// TIA Portal project "SepDuplo" (V16)

(* hardware
DEVICE "S71500/ET200MP station_1"  S7-1500 station
   slot 0: "Rail_0"  Rack  6ES7 590-1***0-0AA0
   slot 1: "PLC_1"  CPU 1512C-1 PN  6ES7 512-1CK00-0AB0  V2.8
      slot 3: "CPU display_1"  6ES7591-1AA00-0AA0
      slot 32768: "PROFINET interface_1"  X1
         slot 32769: "Port_1"  X1 P1
         slot 32770: "Port_2"  X1 P2
      slot 34817: "Virtual CP interface port_1"  Virtual CP interface port  Virtual CP interface port
*)

// ===== PLC "PLC_1"  CPU 1512C-1 PN =====

VAR_GLOBAL   // PLC tag table "Default tag table"
   "alwaysFalse" AT %M0.0 : Bool;
END_VAR

VAR_GLOBAL   // PLC tag table "E_N_Controlavel"
   "FIO_S3" AT %M5.3 : Bool;
   "FIO_PA1" AT %M5.1 : Bool;
   "FIO_PV1" AT %M5.0 : Bool;
   "FIO_S4" AT %M5.5 : Bool;
   "FIO_AT1_Fwd" AT %M5.6 : Bool;
   "FIO_AT1_Rev" AT %M5.7 : Bool;
   "FIO_PA2" AT %M6.0 : Bool;
   "FIO_PV2" AT %M6.1 : Bool;
   "FIO_S5" AT %M6.2 : Bool;
   "FIO_S6" AT %M6.3 : Bool;
   "FIO_AT2_Fwd" AT %M6.4 : Bool;
   "FIO_AT2_Rev" AT %M6.5 : Bool;
END_VAR

VAR_GLOBAL   // PLC tag table "Saidas"
   "FIO_Atuador1" AT %M10.0 : Bool;
   "FIO_Esteira1" AT %M10.1 : Bool;
   "FIO_Esteira2" AT %M10.2 : Bool;
   "FIO_Esteira3" AT %M10.3 : Bool;
   "FIO_Esteira4" AT %M10.4 : Bool;
   "FIO_Atuador2" AT %M10.5 : Bool;
END_VAR

DATA_BLOCK "Eventos"   // DB1
{ S7_Optimized_Access := 'TRUE' }
VERSION : 0.1
   VAR
      PV1_Ev : Bool;
      PA1_Ev : Bool;
      PV2_Ev : Bool;
      PA2_Ev : Bool;
      S3_On_Ev : Bool;
      S3_On_Mirror : Bool;
      S3_Off_Ev : Bool;
      S4_On_Ev : Bool;
      S4_On_Mirror : Bool;
      S4_Off_Ev : Bool;
      AT1_Off_Ev : Bool;
      AT2_Off_Ev : Bool;
      S5_Off_Ev : Bool;
      S6_Off_Ev : Bool;
      AT1_On_Ev : Bool;
      AT2_On_Ev : Bool;
      E1_On_Ev : Bool;
      E1_Off_Ev : Bool;
      E2_On_Ev : Bool;
      E2_Off_Ev : Bool;
      E3_On_Ev : Bool;
      E3_Off_Ev : Bool;
      E4_On_Ev : Bool;
      E4_Off_Ev : Bool;
   END_VAR
BEGIN
END_DATA_BLOCK

DATA_BLOCK "BitsAuxiliares"   // DB2
{ S7_Optimized_Access := 'TRUE' }
VERSION : 0.1
   VAR
      Aux1 : Bool;
      Aux2 : Bool;
      Aux3 : Bool;
      Aux4 : Bool;
      Aux5 : Bool;
      Aux6 : Bool;
      Aux7 : Bool;
      Aux8 : Bool;
      Aux9 : Bool;
      Aux10 : Bool;
      Aux11 : Bool;
      Aux12 : Bool;
   END_VAR
BEGIN
END_DATA_BLOCK

DATA_BLOCK "EstadosSP"   // DB3
{ S7_Optimized_Access := 'TRUE' }
VERSION : 0.1
   VAR
      GS1_1 : Bool := true;
      GS1_2 : Bool;
      GS1_3 : Bool;
      GS2_1 : Bool := true;
      GS2_2 : Bool;
      GS2_3 : Bool;
      GAT1_1 : Bool := true;
      GAT1_2 : Bool;
      GAT2_1 : Bool := true;
      GAT2_2 : Bool;
      GE1_1 : Bool := true;
      GE1_2 : Bool;
      GE2_1 : Bool := true;
      GE2_2 : Bool;
      GE3_1 : Bool := true;
      GE3_2 : Bool;
      GE4_1 : Bool := true;
      GE4_2 : Bool;
      GS5_1 : Bool := true;
      GS6_1 : Bool := true;
   END_VAR
BEGIN
END_DATA_BLOCK

DATA_BLOCK "EstadosSup"   // DB4
{ S7_Optimized_Access := 'TRUE' }
VERSION : 0.1
   VAR
      Sup1_1 : Bool := true;
      Sup1_2 : Bool;
      Sup2_1 : Bool := true;
      Sup2_2 : Bool;
      Sup3_1 : Bool := true;
      Sup3_2 : Bool;
      Sup3_3 : Bool;
      Sup3_4 : Bool;
      Sup4_1 : Bool := true;
      Sup4_2 : Bool;
      Sup4_3 : Bool;
      Sup4_4 : Bool;
      Sup5_1 : Bool := true;
      Sup5_2 : Bool;
      Sup6_1 : Bool := true;
      Sup6_2 : Bool;
      Sup7_1 : Bool := true;
      Sup7_2 : Bool;
      Sup7_3 : Bool;
      Sup8_1 : Bool := true;
      Sup8_2 : Bool;
      Sup8_3 : Bool;
      Sup9_1 : Bool := true;
      Sup9_2 : Bool;
      Sup10_1 : Bool := true;
      Sup10_2 : Bool;
      Sup11_1 : Bool := true;
      Sup11_2 : Bool;
      Sup12_1 : Bool := true;
      Sup12_2 : Bool;
      Sup13_1 : Bool := true;
      Sup13_2 : Bool;
      Sup13_3 : Bool;
      Sup13_4 : Bool;
      Sup13_5 : Bool;
      Sup13_6 : Bool;
      Sup13_7 : Bool;
      Sup13_8 : Bool;
      Sup13_9 : Bool;
      Sup14_1 : Bool := true;
      Sup14_2 : Bool;
      Sup15_1 : Bool := true;
      Sup15_2 : Bool;
   END_VAR
BEGIN
END_DATA_BLOCK

DATA_BLOCK "Des_Eventos"   // DB5
{ S7_Optimized_Access := 'TRUE' }
VERSION : 0.1
   VAR
      d_AT1_On : Bool;
      d_AT2_On : Bool;
      d_E1_On : Bool;
      d_E1_Off : Bool;
      d_E2_On : Bool;
      d_E2_Off : Bool;
      d_E3_On : Bool;
      d_E3_Off : Bool;
      d_E4_On : Bool;
      d_E4_Off : Bool;
   END_VAR
BEGIN
END_DATA_BLOCK

FUNCTION "LeituraEntradas" : Void   // FC2, LAD
TITLE = Leitura das entradas dos eventos não controláveis
{ S7_Optimized_Access := 'TRUE' }
VERSION : 0.1
   VAR_TEMP   // added for the SCL form of the ladder/FBD networks
      _w1 : Bool;
   END_VAR
BEGIN

REGION Network 1: Leitura peça verde 1
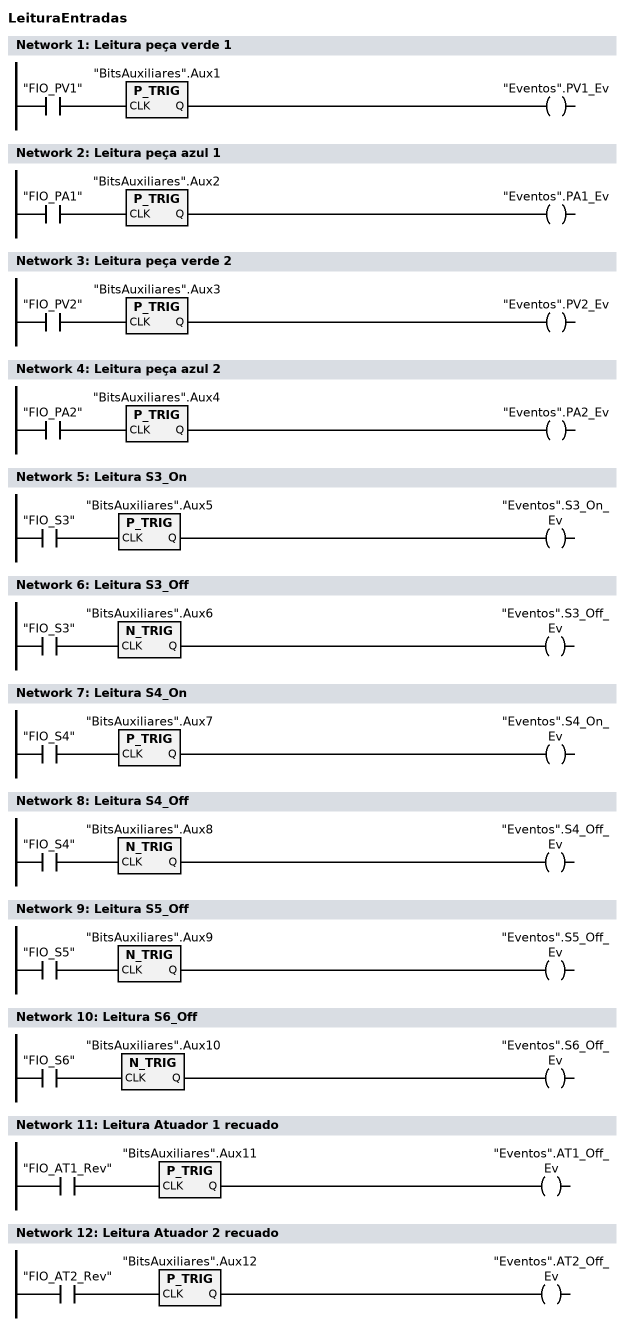
   RUNG wire#powerrail
      Contact( "FIO_PV1" )
      P_Trig( "BitsAuxiliares".Aux1 )
      Coil( "Eventos".PV1_Ev )
   END_RUNG
   // the same network as SCL:
   #_w1 := "FIO_PV1" AND NOT "BitsAuxiliares".Aux1;   // rising edge
   "BitsAuxiliares".Aux1 := "FIO_PV1";
   "Eventos".PV1_Ev := #_w1;
END_REGION

REGION Network 2: Leitura peça azul 1
   RUNG wire#powerrail
      Contact( "FIO_PA1" )
      P_Trig( "BitsAuxiliares".Aux2 )
      Coil( "Eventos".PA1_Ev )
   END_RUNG
   // the same network as SCL:
   #_w1 := "FIO_PA1" AND NOT "BitsAuxiliares".Aux2;   // rising edge
   "BitsAuxiliares".Aux2 := "FIO_PA1";
   "Eventos".PA1_Ev := #_w1;
END_REGION

REGION Network 3: Leitura peça verde 2
   RUNG wire#powerrail
      Contact( "FIO_PV2" )
      P_Trig( "BitsAuxiliares".Aux3 )
      Coil( "Eventos".PV2_Ev )
   END_RUNG
   // the same network as SCL:
   #_w1 := "FIO_PV2" AND NOT "BitsAuxiliares".Aux3;   // rising edge
   "BitsAuxiliares".Aux3 := "FIO_PV2";
   "Eventos".PV2_Ev := #_w1;
END_REGION

REGION Network 4: Leitura peça azul 2
   RUNG wire#powerrail
      Contact( "FIO_PA2" )
      P_Trig( "BitsAuxiliares".Aux4 )
      Coil( "Eventos".PA2_Ev )
   END_RUNG
   // the same network as SCL:
   #_w1 := "FIO_PA2" AND NOT "BitsAuxiliares".Aux4;   // rising edge
   "BitsAuxiliares".Aux4 := "FIO_PA2";
   "Eventos".PA2_Ev := #_w1;
END_REGION

REGION Network 5: Leitura S3_On
   RUNG wire#powerrail
      Contact( "FIO_S3" )
      P_Trig( "BitsAuxiliares".Aux5 )
      Coil( "Eventos".S3_On_Ev )
   END_RUNG
   // the same network as SCL:
   #_w1 := "FIO_S3" AND NOT "BitsAuxiliares".Aux5;   // rising edge
   "BitsAuxiliares".Aux5 := "FIO_S3";
   "Eventos".S3_On_Ev := #_w1;
END_REGION

REGION Network 6: Leitura S3_Off
   RUNG wire#powerrail
      Contact( "FIO_S3" )
      N_Trig( "BitsAuxiliares".Aux6 )
      Coil( "Eventos".S3_Off_Ev )
   END_RUNG
   // the same network as SCL:
   #_w1 := NOT "FIO_S3" AND "BitsAuxiliares".Aux6;   // falling edge
   "BitsAuxiliares".Aux6 := "FIO_S3";
   "Eventos".S3_Off_Ev := #_w1;
END_REGION

REGION Network 7: Leitura S4_On
   RUNG wire#powerrail
      Contact( "FIO_S4" )
      P_Trig( "BitsAuxiliares".Aux7 )
      Coil( "Eventos".S4_On_Ev )
   END_RUNG
   // the same network as SCL:
   #_w1 := "FIO_S4" AND NOT "BitsAuxiliares".Aux7;   // rising edge
   "BitsAuxiliares".Aux7 := "FIO_S4";
   "Eventos".S4_On_Ev := #_w1;
END_REGION

REGION Network 8: Leitura S4_Off
   RUNG wire#powerrail
      Contact( "FIO_S4" )
      N_Trig( "BitsAuxiliares".Aux8 )
      Coil( "Eventos".S4_Off_Ev )
   END_RUNG
   // the same network as SCL:
   #_w1 := NOT "FIO_S4" AND "BitsAuxiliares".Aux8;   // falling edge
   "BitsAuxiliares".Aux8 := "FIO_S4";
   "Eventos".S4_Off_Ev := #_w1;
END_REGION

REGION Network 9: Leitura S5_Off
   RUNG wire#powerrail
      Contact( "FIO_S5" )
      N_Trig( "BitsAuxiliares".Aux9 )
      Coil( "Eventos".S5_Off_Ev )
   END_RUNG
   // the same network as SCL:
   #_w1 := NOT "FIO_S5" AND "BitsAuxiliares".Aux9;   // falling edge
   "BitsAuxiliares".Aux9 := "FIO_S5";
   "Eventos".S5_Off_Ev := #_w1;
END_REGION

REGION Network 10: Leitura S6_Off
   RUNG wire#powerrail
      Contact( "FIO_S6" )
      N_Trig( "BitsAuxiliares".Aux10 )
      Coil( "Eventos".S6_Off_Ev )
   END_RUNG
   // the same network as SCL:
   #_w1 := NOT "FIO_S6" AND "BitsAuxiliares".Aux10;   // falling edge
   "BitsAuxiliares".Aux10 := "FIO_S6";
   "Eventos".S6_Off_Ev := #_w1;
END_REGION

REGION Network 11: Leitura Atuador 1 recuado
   RUNG wire#powerrail
      Contact( "FIO_AT1_Rev" )
      P_Trig( "BitsAuxiliares".Aux11 )
      Coil( "Eventos".AT1_Off_Ev )
   END_RUNG
   // the same network as SCL:
   #_w1 := "FIO_AT1_Rev" AND NOT "BitsAuxiliares".Aux11;   // rising edge
   "BitsAuxiliares".Aux11 := "FIO_AT1_Rev";
   "Eventos".AT1_Off_Ev := #_w1;
END_REGION

REGION Network 12: Leitura Atuador 2 recuado
   RUNG wire#powerrail
      Contact( "FIO_AT2_Rev" )
      P_Trig( "BitsAuxiliares".Aux12 )
      Coil( "Eventos".AT2_Off_Ev )
   END_RUNG
   // the same network as SCL:
   #_w1 := "FIO_AT2_Rev" AND NOT "BitsAuxiliares".Aux12;   // rising edge
   "BitsAuxiliares".Aux12 := "FIO_AT2_Rev";
   "Eventos".AT2_Off_Ev := #_w1;
END_REGION
END_FUNCTION

FUNCTION "At_SP_NaoControlaveis" : Void   // FC3, LAD
TITLE = Atualização dos estados do sistema produto a partir dos eventos não controláveis.
{ S7_Optimized_Access := 'TRUE' }
VERSION : 0.1
BEGIN

REGION Network 1: Modelo de AT1, do estado 2 para o estado 1.
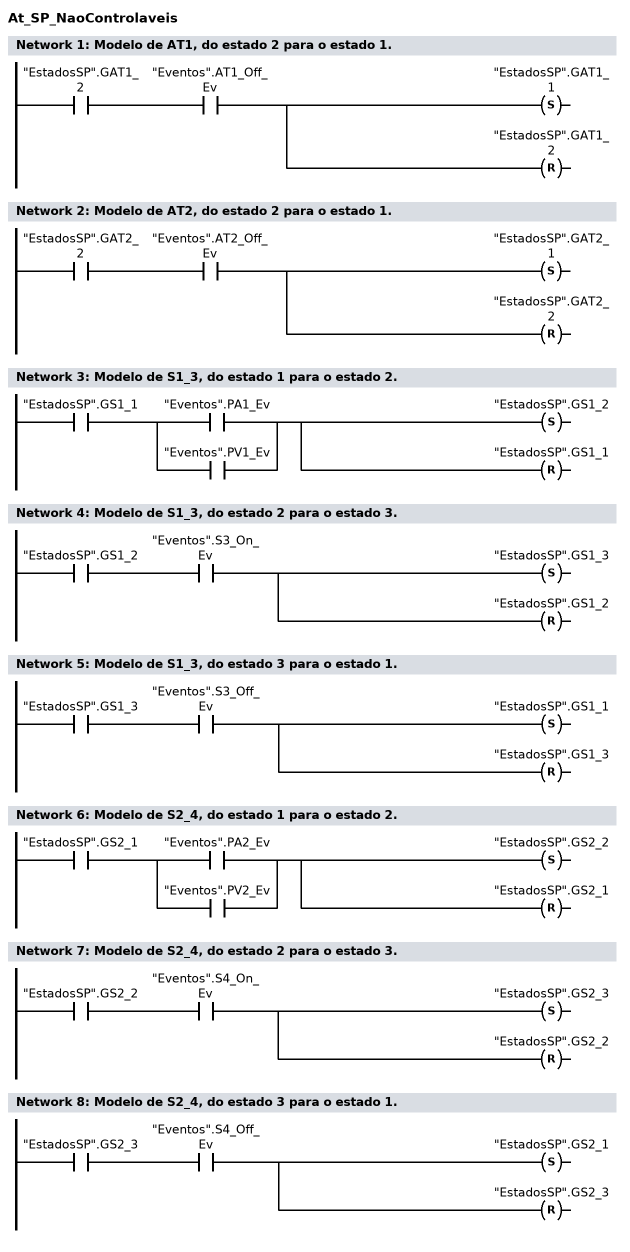
   RUNG wire#powerrail
      Contact( "EstadosSP".GAT1_2 )
      Contact( "Eventos".AT1_Off_Ev )
      wire#w1
      S_Coil( "EstadosSP".GAT1_1 )
   END_RUNG
   RUNG wire#w1
      R_Coil( "EstadosSP".GAT1_2 )
   END_RUNG
   // the same network as SCL:
   IF "EstadosSP".GAT1_2 AND "Eventos".AT1_Off_Ev THEN
       "EstadosSP".GAT1_1 := TRUE;
       "EstadosSP".GAT1_2 := FALSE;
   END_IF;
END_REGION

REGION Network 2: Modelo de AT2, do estado 2 para o estado 1.
   RUNG wire#powerrail
      Contact( "EstadosSP".GAT2_2 )
      Contact( "Eventos".AT2_Off_Ev )
      wire#w1
      S_Coil( "EstadosSP".GAT2_1 )
   END_RUNG
   RUNG wire#w1
      R_Coil( "EstadosSP".GAT2_2 )
   END_RUNG
   // the same network as SCL:
   IF "EstadosSP".GAT2_2 AND "Eventos".AT2_Off_Ev THEN
       "EstadosSP".GAT2_1 := TRUE;
       "EstadosSP".GAT2_2 := FALSE;
   END_IF;
END_REGION

REGION Network 3: Modelo de S1_3, do estado 1 para o estado 2.
   RUNG wire#powerrail
      Contact( "EstadosSP".GS1_1 )
      wire#w1
      Contact( "Eventos".PA1_Ev )
      wire#w2
      S_Coil( "EstadosSP".GS1_2 )
   END_RUNG
   RUNG wire#w1
      Contact( "Eventos".PV1_Ev )
   END_RUNG wire#w2
   RUNG wire#w2
      R_Coil( "EstadosSP".GS1_1 )
   END_RUNG
   // the same network as SCL:
   IF "EstadosSP".GS1_1 AND ("Eventos".PA1_Ev OR "Eventos".PV1_Ev) THEN
       "EstadosSP".GS1_2 := TRUE;
       "EstadosSP".GS1_1 := FALSE;
   END_IF;
END_REGION

REGION Network 4: Modelo de S1_3, do estado 2 para o estado 3.
   RUNG wire#powerrail
      Contact( "EstadosSP".GS1_2 )
      Contact( "Eventos".S3_On_Ev )
      wire#w1
      S_Coil( "EstadosSP".GS1_3 )
   END_RUNG
   RUNG wire#w1
      R_Coil( "EstadosSP".GS1_2 )
   END_RUNG
   // the same network as SCL:
   IF "EstadosSP".GS1_2 AND "Eventos".S3_On_Ev THEN
       "EstadosSP".GS1_3 := TRUE;
       "EstadosSP".GS1_2 := FALSE;
   END_IF;
END_REGION

REGION Network 5: Modelo de S1_3, do estado 3 para o estado 1.
   RUNG wire#powerrail
      Contact( "EstadosSP".GS1_3 )
      Contact( "Eventos".S3_Off_Ev )
      wire#w1
      S_Coil( "EstadosSP".GS1_1 )
   END_RUNG
   RUNG wire#w1
      R_Coil( "EstadosSP".GS1_3 )
   END_RUNG
   // the same network as SCL:
   IF "EstadosSP".GS1_3 AND "Eventos".S3_Off_Ev THEN
       "EstadosSP".GS1_1 := TRUE;
       "EstadosSP".GS1_3 := FALSE;
   END_IF;
END_REGION

REGION Network 6: Modelo de S2_4, do estado 1 para o estado 2.
   RUNG wire#powerrail
      Contact( "EstadosSP".GS2_1 )
      wire#w1
      Contact( "Eventos".PA2_Ev )
      wire#w2
      S_Coil( "EstadosSP".GS2_2 )
   END_RUNG
   RUNG wire#w1
      Contact( "Eventos".PV2_Ev )
   END_RUNG wire#w2
   RUNG wire#w2
      R_Coil( "EstadosSP".GS2_1 )
   END_RUNG
   // the same network as SCL:
   IF "EstadosSP".GS2_1 AND ("Eventos".PA2_Ev OR "Eventos".PV2_Ev) THEN
       "EstadosSP".GS2_2 := TRUE;
       "EstadosSP".GS2_1 := FALSE;
   END_IF;
END_REGION

REGION Network 7: Modelo de S2_4, do estado 2 para o estado 3.
   RUNG wire#powerrail
      Contact( "EstadosSP".GS2_2 )
      Contact( "Eventos".S4_On_Ev )
      wire#w1
      S_Coil( "EstadosSP".GS2_3 )
   END_RUNG
   RUNG wire#w1
      R_Coil( "EstadosSP".GS2_2 )
   END_RUNG
   // the same network as SCL:
   IF "EstadosSP".GS2_2 AND "Eventos".S4_On_Ev THEN
       "EstadosSP".GS2_3 := TRUE;
       "EstadosSP".GS2_2 := FALSE;
   END_IF;
END_REGION

REGION Network 8: Modelo de S2_4, do estado 3 para o estado 1.
   RUNG wire#powerrail
      Contact( "EstadosSP".GS2_3 )
      Contact( "Eventos".S4_Off_Ev )
      wire#w1
      S_Coil( "EstadosSP".GS2_1 )
   END_RUNG
   RUNG wire#w1
      R_Coil( "EstadosSP".GS2_3 )
   END_RUNG
   // the same network as SCL:
   IF "EstadosSP".GS2_3 AND "Eventos".S4_Off_Ev THEN
       "EstadosSP".GS2_1 := TRUE;
       "EstadosSP".GS2_3 := FALSE;
   END_IF;
END_REGION
END_FUNCTION

FUNCTION "At_Sup_NaoControlaveis" : Void   // FC4, LAD
TITLE = Atualização dos estados dos supervisores reduzidos, devido a eventos não controláveis
{ S7_Optimized_Access := 'TRUE' }
VERSION : 0.1
   VAR_TEMP   // added for the SCL form of the ladder/FBD networks
      _w1 : Bool;
   END_VAR
BEGIN

REGION Network 1: Atualização do supervisor 1, estado 1 para estado 2.
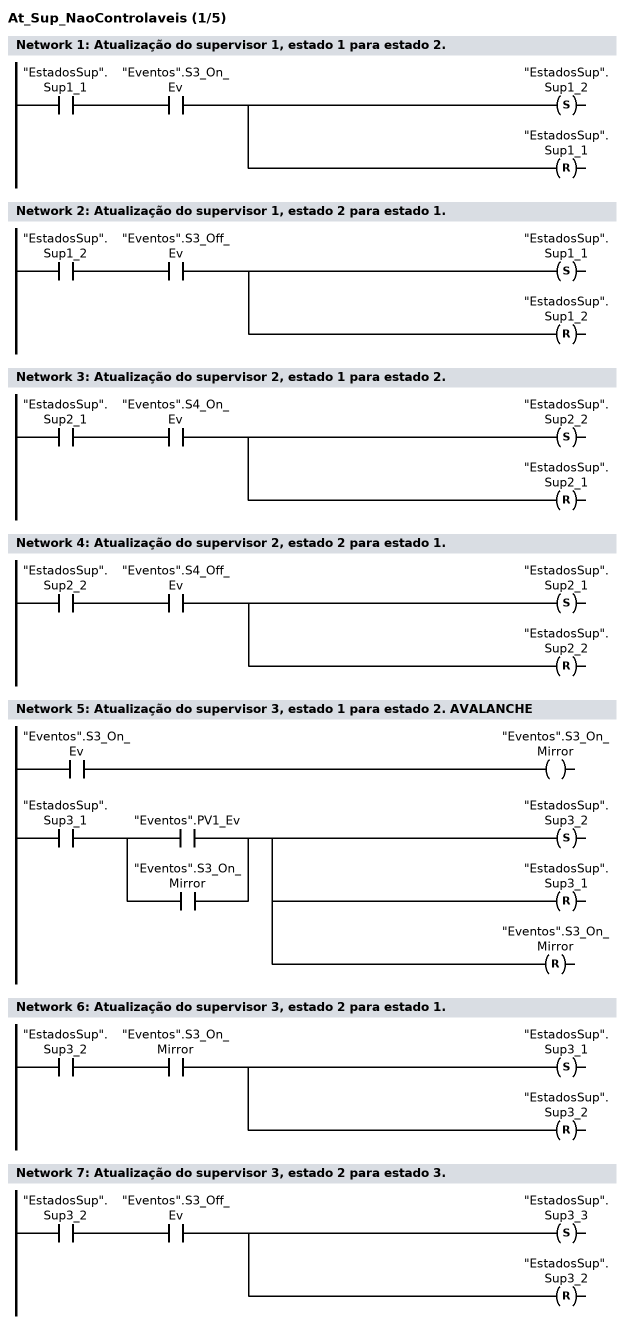
   RUNG wire#powerrail
      Contact( "EstadosSup".Sup1_1 )
      Contact( "Eventos".S3_On_Ev )
      wire#w1
      S_Coil( "EstadosSup".Sup1_2 )
   END_RUNG
   RUNG wire#w1
      R_Coil( "EstadosSup".Sup1_1 )
   END_RUNG
   // the same network as SCL:
   IF "EstadosSup".Sup1_1 AND "Eventos".S3_On_Ev THEN
       "EstadosSup".Sup1_2 := TRUE;
       "EstadosSup".Sup1_1 := FALSE;
   END_IF;
END_REGION

REGION Network 2: Atualização do supervisor 1, estado 2 para estado 1.
   RUNG wire#powerrail
      Contact( "EstadosSup".Sup1_2 )
      Contact( "Eventos".S3_Off_Ev )
      wire#w1
      S_Coil( "EstadosSup".Sup1_1 )
   END_RUNG
   RUNG wire#w1
      R_Coil( "EstadosSup".Sup1_2 )
   END_RUNG
   // the same network as SCL:
   IF "EstadosSup".Sup1_2 AND "Eventos".S3_Off_Ev THEN
       "EstadosSup".Sup1_1 := TRUE;
       "EstadosSup".Sup1_2 := FALSE;
   END_IF;
END_REGION

REGION Network 3: Atualização do supervisor 2, estado 1 para estado 2.
   RUNG wire#powerrail
      Contact( "EstadosSup".Sup2_1 )
      Contact( "Eventos".S4_On_Ev )
      wire#w1
      S_Coil( "EstadosSup".Sup2_2 )
   END_RUNG
   RUNG wire#w1
      R_Coil( "EstadosSup".Sup2_1 )
   END_RUNG
   // the same network as SCL:
   IF "EstadosSup".Sup2_1 AND "Eventos".S4_On_Ev THEN
       "EstadosSup".Sup2_2 := TRUE;
       "EstadosSup".Sup2_1 := FALSE;
   END_IF;
END_REGION

REGION Network 4: Atualização do supervisor 2, estado 2 para estado 1.
   RUNG wire#powerrail
      Contact( "EstadosSup".Sup2_2 )
      Contact( "Eventos".S4_Off_Ev )
      wire#w1
      S_Coil( "EstadosSup".Sup2_1 )
   END_RUNG
   RUNG wire#w1
      R_Coil( "EstadosSup".Sup2_2 )
   END_RUNG
   // the same network as SCL:
   IF "EstadosSup".Sup2_2 AND "Eventos".S4_Off_Ev THEN
       "EstadosSup".Sup2_1 := TRUE;
       "EstadosSup".Sup2_2 := FALSE;
   END_IF;
END_REGION

REGION Network 5: Atualização do supervisor 3, estado 1 para estado 2. AVALANCHE
   RUNG wire#powerrail
      Contact( "Eventos".S3_On_Ev )
      Coil( "Eventos".S3_On_Mirror )
   END_RUNG
   RUNG wire#powerrail
      Contact( "EstadosSup".Sup3_1 )
      wire#w1
      Contact( "Eventos".PV1_Ev )
      wire#w2
      S_Coil( "EstadosSup".Sup3_2 )
   END_RUNG
   RUNG wire#w1
      Contact( "Eventos".S3_On_Mirror )
   END_RUNG wire#w2
   RUNG wire#w2
      R_Coil( "EstadosSup".Sup3_1 )
   END_RUNG
   RUNG wire#w2
      R_Coil( "Eventos".S3_On_Mirror )
   END_RUNG
   // the same network as SCL:
   "Eventos".S3_On_Mirror := "Eventos".S3_On_Ev;
   IF "EstadosSup".Sup3_1 AND ("Eventos".PV1_Ev OR "Eventos".S3_On_Mirror) THEN
       "EstadosSup".Sup3_2 := TRUE;
   END_IF;
   #_w1 := "EstadosSup".Sup3_1 AND ("Eventos".PV1_Ev OR "Eventos".S3_On_Mirror);
   IF #_w1 THEN
       "EstadosSup".Sup3_1 := FALSE;
       "Eventos".S3_On_Mirror := FALSE;
   END_IF;
END_REGION

REGION Network 6: Atualização do supervisor 3, estado 2 para estado 1.
   RUNG wire#powerrail
      Contact( "EstadosSup".Sup3_2 )
      Contact( "Eventos".S3_On_Mirror )
      wire#w1
      S_Coil( "EstadosSup".Sup3_1 )
   END_RUNG
   RUNG wire#w1
      R_Coil( "EstadosSup".Sup3_2 )
   END_RUNG
   // the same network as SCL:
   IF "EstadosSup".Sup3_2 AND "Eventos".S3_On_Mirror THEN
       "EstadosSup".Sup3_1 := TRUE;
       "EstadosSup".Sup3_2 := FALSE;
   END_IF;
END_REGION

REGION Network 7: Atualização do supervisor 3, estado 2 para estado 3.
   RUNG wire#powerrail
      Contact( "EstadosSup".Sup3_2 )
      Contact( "Eventos".S3_Off_Ev )
      wire#w1
      S_Coil( "EstadosSup".Sup3_3 )
   END_RUNG
   RUNG wire#w1
      R_Coil( "EstadosSup".Sup3_2 )
   END_RUNG
   // the same network as SCL:
   IF "EstadosSup".Sup3_2 AND "Eventos".S3_Off_Ev THEN
       "EstadosSup".Sup3_3 := TRUE;
       "EstadosSup".Sup3_2 := FALSE;
   END_IF;
END_REGION

REGION Network 8: Atualização do supervisor 3, estado 3 para estado 4.
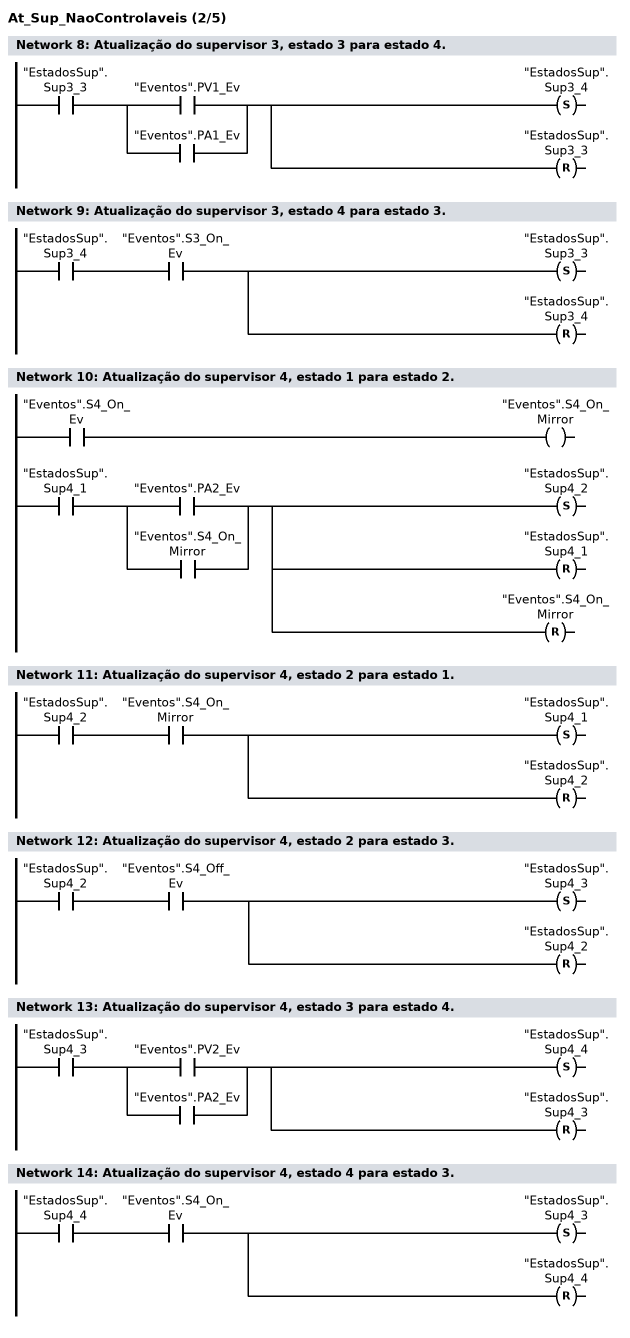
   RUNG wire#powerrail
      Contact( "EstadosSup".Sup3_3 )
      wire#w1
      Contact( "Eventos".PV1_Ev )
      wire#w2
      S_Coil( "EstadosSup".Sup3_4 )
   END_RUNG
   RUNG wire#w1
      Contact( "Eventos".PA1_Ev )
   END_RUNG wire#w2
   RUNG wire#w2
      R_Coil( "EstadosSup".Sup3_3 )
   END_RUNG
   // the same network as SCL:
   IF "EstadosSup".Sup3_3 AND ("Eventos".PV1_Ev OR "Eventos".PA1_Ev) THEN
       "EstadosSup".Sup3_4 := TRUE;
       "EstadosSup".Sup3_3 := FALSE;
   END_IF;
END_REGION

REGION Network 9: Atualização do supervisor 3, estado 4 para estado 3.
   RUNG wire#powerrail
      Contact( "EstadosSup".Sup3_4 )
      Contact( "Eventos".S3_On_Ev )
      wire#w1
      S_Coil( "EstadosSup".Sup3_3 )
   END_RUNG
   RUNG wire#w1
      R_Coil( "EstadosSup".Sup3_4 )
   END_RUNG
   // the same network as SCL:
   IF "EstadosSup".Sup3_4 AND "Eventos".S3_On_Ev THEN
       "EstadosSup".Sup3_3 := TRUE;
       "EstadosSup".Sup3_4 := FALSE;
   END_IF;
END_REGION

REGION Network 10: Atualização do supervisor 4, estado 1 para estado 2.
   RUNG wire#powerrail
      Contact( "Eventos".S4_On_Ev )
      Coil( "Eventos".S4_On_Mirror )
   END_RUNG
   RUNG wire#powerrail
      Contact( "EstadosSup".Sup4_1 )
      wire#w1
      Contact( "Eventos".PA2_Ev )
      wire#w2
      S_Coil( "EstadosSup".Sup4_2 )
   END_RUNG
   RUNG wire#w1
      Contact( "Eventos".S4_On_Mirror )
   END_RUNG wire#w2
   RUNG wire#w2
      R_Coil( "EstadosSup".Sup4_1 )
   END_RUNG
   RUNG wire#w2
      R_Coil( "Eventos".S4_On_Mirror )
   END_RUNG
   // the same network as SCL:
   "Eventos".S4_On_Mirror := "Eventos".S4_On_Ev;
   IF "EstadosSup".Sup4_1 AND ("Eventos".PA2_Ev OR "Eventos".S4_On_Mirror) THEN
       "EstadosSup".Sup4_2 := TRUE;
   END_IF;
   #_w1 := "EstadosSup".Sup4_1 AND ("Eventos".PA2_Ev OR "Eventos".S4_On_Mirror);
   IF #_w1 THEN
       "EstadosSup".Sup4_1 := FALSE;
       "Eventos".S4_On_Mirror := FALSE;
   END_IF;
END_REGION

REGION Network 11: Atualização do supervisor 4, estado 2 para estado 1.
   RUNG wire#powerrail
      Contact( "EstadosSup".Sup4_2 )
      Contact( "Eventos".S4_On_Mirror )
      wire#w1
      S_Coil( "EstadosSup".Sup4_1 )
   END_RUNG
   RUNG wire#w1
      R_Coil( "EstadosSup".Sup4_2 )
   END_RUNG
   // the same network as SCL:
   IF "EstadosSup".Sup4_2 AND "Eventos".S4_On_Mirror THEN
       "EstadosSup".Sup4_1 := TRUE;
       "EstadosSup".Sup4_2 := FALSE;
   END_IF;
END_REGION

REGION Network 12: Atualização do supervisor 4, estado 2 para estado 3.
   RUNG wire#powerrail
      Contact( "EstadosSup".Sup4_2 )
      Contact( "Eventos".S4_Off_Ev )
      wire#w1
      S_Coil( "EstadosSup".Sup4_3 )
   END_RUNG
   RUNG wire#w1
      R_Coil( "EstadosSup".Sup4_2 )
   END_RUNG
   // the same network as SCL:
   IF "EstadosSup".Sup4_2 AND "Eventos".S4_Off_Ev THEN
       "EstadosSup".Sup4_3 := TRUE;
       "EstadosSup".Sup4_2 := FALSE;
   END_IF;
END_REGION

REGION Network 13: Atualização do supervisor 4, estado 3 para estado 4.
   RUNG wire#powerrail
      Contact( "EstadosSup".Sup4_3 )
      wire#w1
      Contact( "Eventos".PV2_Ev )
      wire#w2
      S_Coil( "EstadosSup".Sup4_4 )
   END_RUNG
   RUNG wire#w1
      Contact( "Eventos".PA2_Ev )
   END_RUNG wire#w2
   RUNG wire#w2
      R_Coil( "EstadosSup".Sup4_3 )
   END_RUNG
   // the same network as SCL:
   IF "EstadosSup".Sup4_3 AND ("Eventos".PV2_Ev OR "Eventos".PA2_Ev) THEN
       "EstadosSup".Sup4_4 := TRUE;
       "EstadosSup".Sup4_3 := FALSE;
   END_IF;
END_REGION

REGION Network 14: Atualização do supervisor 4, estado 4 para estado 3.
   RUNG wire#powerrail
      Contact( "EstadosSup".Sup4_4 )
      Contact( "Eventos".S4_On_Ev )
      wire#w1
      S_Coil( "EstadosSup".Sup4_3 )
   END_RUNG
   RUNG wire#w1
      R_Coil( "EstadosSup".Sup4_4 )
   END_RUNG
   // the same network as SCL:
   IF "EstadosSup".Sup4_4 AND "Eventos".S4_On_Ev THEN
       "EstadosSup".Sup4_3 := TRUE;
       "EstadosSup".Sup4_4 := FALSE;
   END_IF;
END_REGION

REGION Network 15: Atualização do supervisor 5, estado 2 para estado 1.
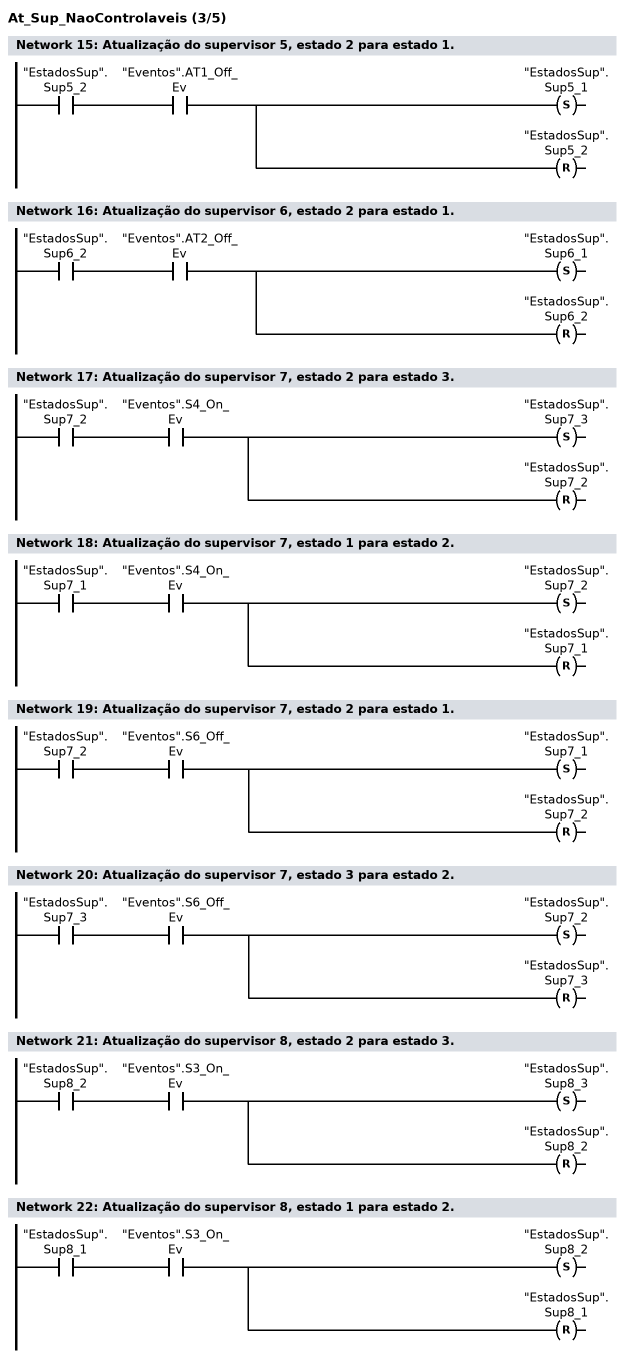
   RUNG wire#powerrail
      Contact( "EstadosSup".Sup5_2 )
      Contact( "Eventos".AT1_Off_Ev )
      wire#w1
      S_Coil( "EstadosSup".Sup5_1 )
   END_RUNG
   RUNG wire#w1
      R_Coil( "EstadosSup".Sup5_2 )
   END_RUNG
   // the same network as SCL:
   IF "EstadosSup".Sup5_2 AND "Eventos".AT1_Off_Ev THEN
       "EstadosSup".Sup5_1 := TRUE;
       "EstadosSup".Sup5_2 := FALSE;
   END_IF;
END_REGION

REGION Network 16: Atualização do supervisor 6, estado 2 para estado 1.
   RUNG wire#powerrail
      Contact( "EstadosSup".Sup6_2 )
      Contact( "Eventos".AT2_Off_Ev )
      wire#w1
      S_Coil( "EstadosSup".Sup6_1 )
   END_RUNG
   RUNG wire#w1
      R_Coil( "EstadosSup".Sup6_2 )
   END_RUNG
   // the same network as SCL:
   IF "EstadosSup".Sup6_2 AND "Eventos".AT2_Off_Ev THEN
       "EstadosSup".Sup6_1 := TRUE;
       "EstadosSup".Sup6_2 := FALSE;
   END_IF;
END_REGION

REGION Network 17: Atualização do supervisor 7, estado 2 para estado 3.
   RUNG wire#powerrail
      Contact( "EstadosSup".Sup7_2 )
      Contact( "Eventos".S4_On_Ev )
      wire#w1
      S_Coil( "EstadosSup".Sup7_3 )
   END_RUNG
   RUNG wire#w1
      R_Coil( "EstadosSup".Sup7_2 )
   END_RUNG
   // the same network as SCL:
   IF "EstadosSup".Sup7_2 AND "Eventos".S4_On_Ev THEN
       "EstadosSup".Sup7_3 := TRUE;
       "EstadosSup".Sup7_2 := FALSE;
   END_IF;
END_REGION

REGION Network 18: Atualização do supervisor 7, estado 1 para estado 2.
   RUNG wire#powerrail
      Contact( "EstadosSup".Sup7_1 )
      Contact( "Eventos".S4_On_Ev )
      wire#w1
      S_Coil( "EstadosSup".Sup7_2 )
   END_RUNG
   RUNG wire#w1
      R_Coil( "EstadosSup".Sup7_1 )
   END_RUNG
   // the same network as SCL:
   IF "EstadosSup".Sup7_1 AND "Eventos".S4_On_Ev THEN
       "EstadosSup".Sup7_2 := TRUE;
       "EstadosSup".Sup7_1 := FALSE;
   END_IF;
END_REGION

REGION Network 19: Atualização do supervisor 7, estado 2 para estado 1.
   RUNG wire#powerrail
      Contact( "EstadosSup".Sup7_2 )
      Contact( "Eventos".S6_Off_Ev )
      wire#w1
      S_Coil( "EstadosSup".Sup7_1 )
   END_RUNG
   RUNG wire#w1
      R_Coil( "EstadosSup".Sup7_2 )
   END_RUNG
   // the same network as SCL:
   IF "EstadosSup".Sup7_2 AND "Eventos".S6_Off_Ev THEN
       "EstadosSup".Sup7_1 := TRUE;
       "EstadosSup".Sup7_2 := FALSE;
   END_IF;
END_REGION

REGION Network 20: Atualização do supervisor 7, estado 3 para estado 2.
   RUNG wire#powerrail
      Contact( "EstadosSup".Sup7_3 )
      Contact( "Eventos".S6_Off_Ev )
      wire#w1
      S_Coil( "EstadosSup".Sup7_2 )
   END_RUNG
   RUNG wire#w1
      R_Coil( "EstadosSup".Sup7_3 )
   END_RUNG
   // the same network as SCL:
   IF "EstadosSup".Sup7_3 AND "Eventos".S6_Off_Ev THEN
       "EstadosSup".Sup7_2 := TRUE;
       "EstadosSup".Sup7_3 := FALSE;
   END_IF;
END_REGION

REGION Network 21: Atualização do supervisor 8, estado 2 para estado 3.
   RUNG wire#powerrail
      Contact( "EstadosSup".Sup8_2 )
      Contact( "Eventos".S3_On_Ev )
      wire#w1
      S_Coil( "EstadosSup".Sup8_3 )
   END_RUNG
   RUNG wire#w1
      R_Coil( "EstadosSup".Sup8_2 )
   END_RUNG
   // the same network as SCL:
   IF "EstadosSup".Sup8_2 AND "Eventos".S3_On_Ev THEN
       "EstadosSup".Sup8_3 := TRUE;
       "EstadosSup".Sup8_2 := FALSE;
   END_IF;
END_REGION

REGION Network 22: Atualização do supervisor 8, estado 1 para estado 2.
   RUNG wire#powerrail
      Contact( "EstadosSup".Sup8_1 )
      Contact( "Eventos".S3_On_Ev )
      wire#w1
      S_Coil( "EstadosSup".Sup8_2 )
   END_RUNG
   RUNG wire#w1
      R_Coil( "EstadosSup".Sup8_1 )
   END_RUNG
   // the same network as SCL:
   IF "EstadosSup".Sup8_1 AND "Eventos".S3_On_Ev THEN
       "EstadosSup".Sup8_2 := TRUE;
       "EstadosSup".Sup8_1 := FALSE;
   END_IF;
END_REGION

REGION Network 23: Atualização do supervisor 8, estado 2 para estado 1.
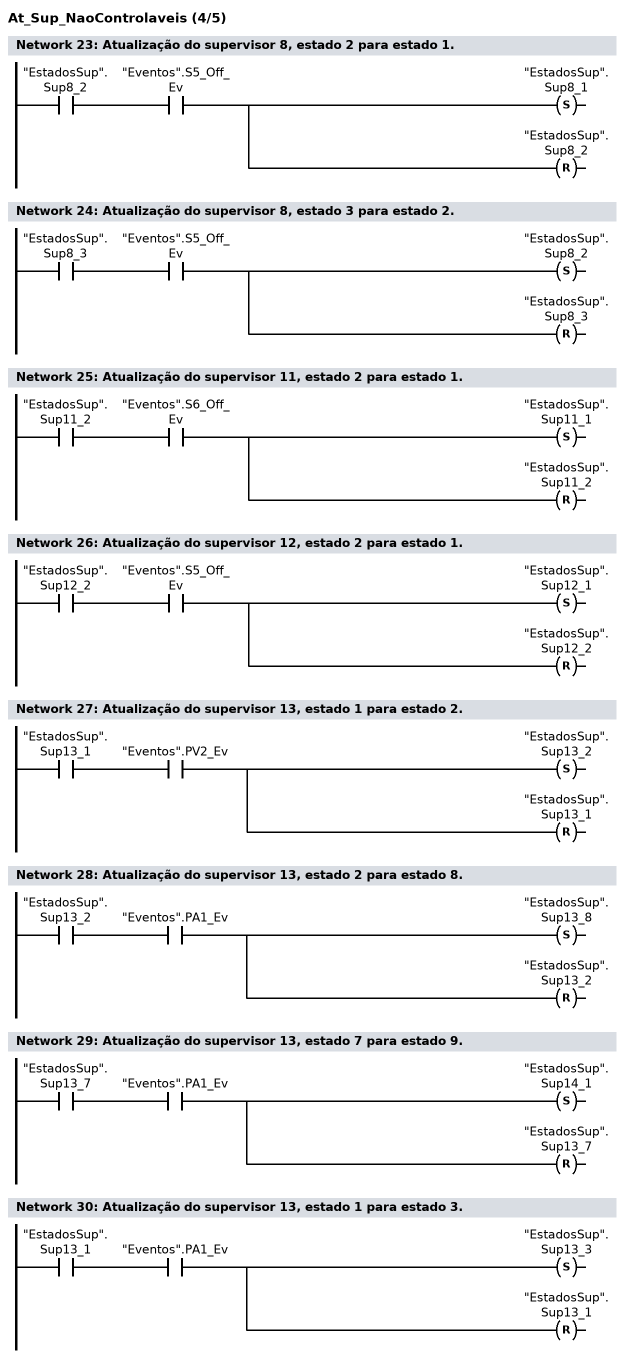
   RUNG wire#powerrail
      Contact( "EstadosSup".Sup8_2 )
      Contact( "Eventos".S5_Off_Ev )
      wire#w1
      S_Coil( "EstadosSup".Sup8_1 )
   END_RUNG
   RUNG wire#w1
      R_Coil( "EstadosSup".Sup8_2 )
   END_RUNG
   // the same network as SCL:
   IF "EstadosSup".Sup8_2 AND "Eventos".S5_Off_Ev THEN
       "EstadosSup".Sup8_1 := TRUE;
       "EstadosSup".Sup8_2 := FALSE;
   END_IF;
END_REGION

REGION Network 24: Atualização do supervisor 8, estado 3 para estado 2.
   RUNG wire#powerrail
      Contact( "EstadosSup".Sup8_3 )
      Contact( "Eventos".S5_Off_Ev )
      wire#w1
      S_Coil( "EstadosSup".Sup8_2 )
   END_RUNG
   RUNG wire#w1
      R_Coil( "EstadosSup".Sup8_3 )
   END_RUNG
   // the same network as SCL:
   IF "EstadosSup".Sup8_3 AND "Eventos".S5_Off_Ev THEN
       "EstadosSup".Sup8_2 := TRUE;
       "EstadosSup".Sup8_3 := FALSE;
   END_IF;
END_REGION

REGION Network 25: Atualização do supervisor 11, estado 2 para estado 1.
   RUNG wire#powerrail
      Contact( "EstadosSup".Sup11_2 )
      Contact( "Eventos".S6_Off_Ev )
      wire#w1
      S_Coil( "EstadosSup".Sup11_1 )
   END_RUNG
   RUNG wire#w1
      R_Coil( "EstadosSup".Sup11_2 )
   END_RUNG
   // the same network as SCL:
   IF "EstadosSup".Sup11_2 AND "Eventos".S6_Off_Ev THEN
       "EstadosSup".Sup11_1 := TRUE;
       "EstadosSup".Sup11_2 := FALSE;
   END_IF;
END_REGION

REGION Network 26: Atualização do supervisor 12, estado 2 para estado 1.
   RUNG wire#powerrail
      Contact( "EstadosSup".Sup12_2 )
      Contact( "Eventos".S5_Off_Ev )
      wire#w1
      S_Coil( "EstadosSup".Sup12_1 )
   END_RUNG
   RUNG wire#w1
      R_Coil( "EstadosSup".Sup12_2 )
   END_RUNG
   // the same network as SCL:
   IF "EstadosSup".Sup12_2 AND "Eventos".S5_Off_Ev THEN
       "EstadosSup".Sup12_1 := TRUE;
       "EstadosSup".Sup12_2 := FALSE;
   END_IF;
END_REGION

REGION Network 27: Atualização do supervisor 13, estado 1 para estado 2.
   RUNG wire#powerrail
      Contact( "EstadosSup".Sup13_1 )
      Contact( "Eventos".PV2_Ev )
      wire#w1
      S_Coil( "EstadosSup".Sup13_2 )
   END_RUNG
   RUNG wire#w1
      R_Coil( "EstadosSup".Sup13_1 )
   END_RUNG
   // the same network as SCL:
   IF "EstadosSup".Sup13_1 AND "Eventos".PV2_Ev THEN
       "EstadosSup".Sup13_2 := TRUE;
       "EstadosSup".Sup13_1 := FALSE;
   END_IF;
END_REGION

REGION Network 28: Atualização do supervisor 13, estado 2 para estado 8.
   RUNG wire#powerrail
      Contact( "EstadosSup".Sup13_2 )
      Contact( "Eventos".PA1_Ev )
      wire#w1
      S_Coil( "EstadosSup".Sup13_8 )
   END_RUNG
   RUNG wire#w1
      R_Coil( "EstadosSup".Sup13_2 )
   END_RUNG
   // the same network as SCL:
   IF "EstadosSup".Sup13_2 AND "Eventos".PA1_Ev THEN
       "EstadosSup".Sup13_8 := TRUE;
       "EstadosSup".Sup13_2 := FALSE;
   END_IF;
END_REGION

REGION Network 29: Atualização do supervisor 13, estado 7 para estado 9.
   RUNG wire#powerrail
      Contact( "EstadosSup".Sup13_7 )
      Contact( "Eventos".PA1_Ev )
      wire#w1
      S_Coil( "EstadosSup".Sup14_1 )
   END_RUNG
   RUNG wire#w1
      R_Coil( "EstadosSup".Sup13_7 )
   END_RUNG
   // the same network as SCL:
   IF "EstadosSup".Sup13_7 AND "Eventos".PA1_Ev THEN
       "EstadosSup".Sup14_1 := TRUE;
       "EstadosSup".Sup13_7 := FALSE;
   END_IF;
END_REGION

REGION Network 30: Atualização do supervisor 13, estado 1 para estado 3.
   RUNG wire#powerrail
      Contact( "EstadosSup".Sup13_1 )
      Contact( "Eventos".PA1_Ev )
      wire#w1
      S_Coil( "EstadosSup".Sup13_3 )
   END_RUNG
   RUNG wire#w1
      R_Coil( "EstadosSup".Sup13_1 )
   END_RUNG
   // the same network as SCL:
   IF "EstadosSup".Sup13_1 AND "Eventos".PA1_Ev THEN
       "EstadosSup".Sup13_3 := TRUE;
       "EstadosSup".Sup13_1 := FALSE;
   END_IF;
END_REGION

REGION Network 31: Atualização do supervisor 13, estado 3 para estado 4.
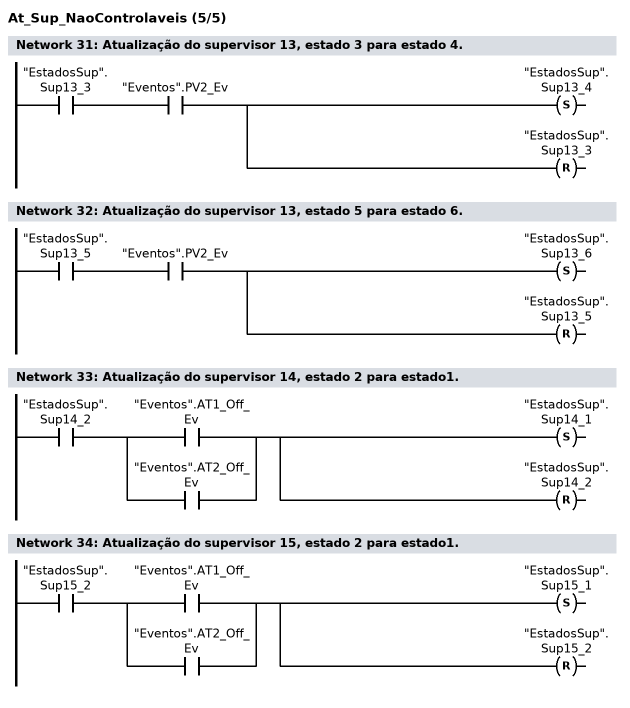
   RUNG wire#powerrail
      Contact( "EstadosSup".Sup13_3 )
      Contact( "Eventos".PV2_Ev )
      wire#w1
      S_Coil( "EstadosSup".Sup13_4 )
   END_RUNG
   RUNG wire#w1
      R_Coil( "EstadosSup".Sup13_3 )
   END_RUNG
   // the same network as SCL:
   IF "EstadosSup".Sup13_3 AND "Eventos".PV2_Ev THEN
       "EstadosSup".Sup13_4 := TRUE;
       "EstadosSup".Sup13_3 := FALSE;
   END_IF;
END_REGION

REGION Network 32: Atualização do supervisor 13, estado 5 para estado 6.
   RUNG wire#powerrail
      Contact( "EstadosSup".Sup13_5 )
      Contact( "Eventos".PV2_Ev )
      wire#w1
      S_Coil( "EstadosSup".Sup13_6 )
   END_RUNG
   RUNG wire#w1
      R_Coil( "EstadosSup".Sup13_5 )
   END_RUNG
   // the same network as SCL:
   IF "EstadosSup".Sup13_5 AND "Eventos".PV2_Ev THEN
       "EstadosSup".Sup13_6 := TRUE;
       "EstadosSup".Sup13_5 := FALSE;
   END_IF;
END_REGION

REGION Network 33: Atualização do supervisor 14, estado 2 para estado1.
   RUNG wire#powerrail
      Contact( "EstadosSup".Sup14_2 )
      wire#w1
      Contact( "Eventos".AT1_Off_Ev )
      wire#w2
      S_Coil( "EstadosSup".Sup14_1 )
   END_RUNG
   RUNG wire#w1
      Contact( "Eventos".AT2_Off_Ev )
   END_RUNG wire#w2
   RUNG wire#w2
      R_Coil( "EstadosSup".Sup14_2 )
   END_RUNG
   // the same network as SCL:
   IF "EstadosSup".Sup14_2 AND ("Eventos".AT1_Off_Ev OR "Eventos".AT2_Off_Ev) THEN
       "EstadosSup".Sup14_1 := TRUE;
       "EstadosSup".Sup14_2 := FALSE;
   END_IF;
END_REGION

REGION Network 34: Atualização do supervisor 15, estado 2 para estado1.
   RUNG wire#powerrail
      Contact( "EstadosSup".Sup15_2 )
      wire#w1
      Contact( "Eventos".AT1_Off_Ev )
      wire#w2
      S_Coil( "EstadosSup".Sup15_1 )
   END_RUNG
   RUNG wire#w1
      Contact( "Eventos".AT2_Off_Ev )
   END_RUNG wire#w2
   RUNG wire#w2
      R_Coil( "EstadosSup".Sup15_2 )
   END_RUNG
   // the same network as SCL:
   IF "EstadosSup".Sup15_2 AND ("Eventos".AT1_Off_Ev OR "Eventos".AT2_Off_Ev) THEN
       "EstadosSup".Sup15_1 := TRUE;
       "EstadosSup".Sup15_2 := FALSE;
   END_IF;
END_REGION
END_FUNCTION

FUNCTION "Des_EventosControlaveis" : Void   // FC5, LAD
TITLE = Desativação dos eventos controláveis
{ S7_Optimized_Access := 'TRUE' }
VERSION : 0.1
BEGIN

REGION Network 1: Desabilita o avanço atuador 1
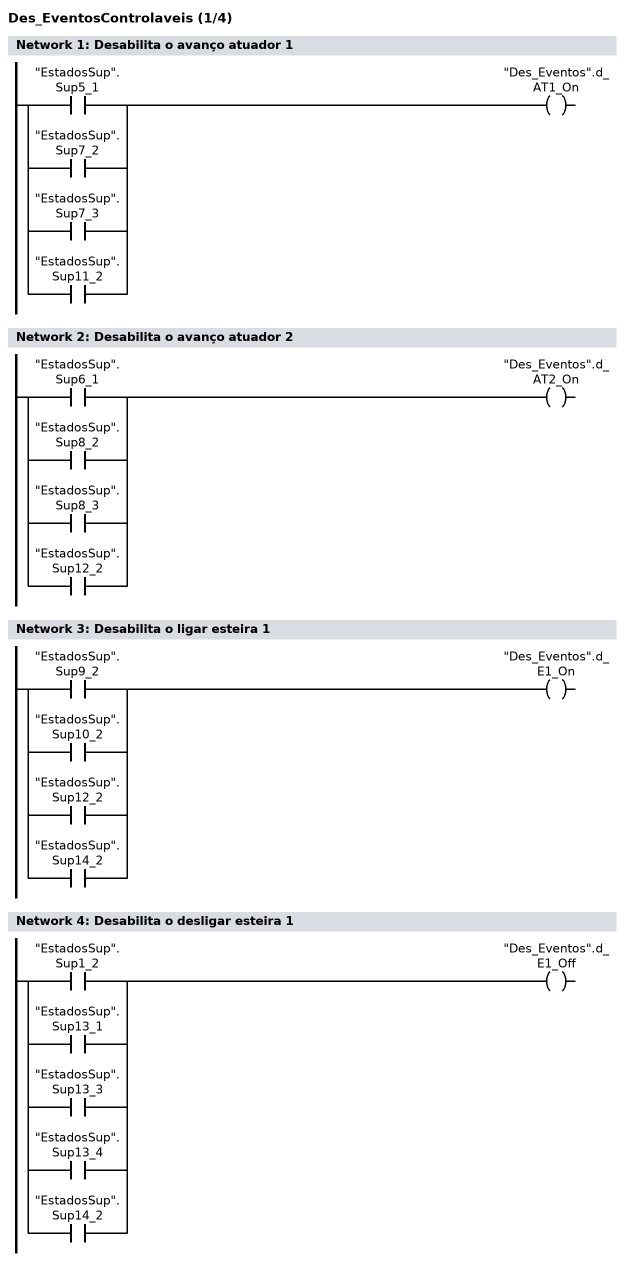
   RUNG wire#powerrail
      Contact( "EstadosSup".Sup5_1 )
      wire#w1
      Coil( "Des_Eventos".d_AT1_On )
   END_RUNG
   RUNG wire#powerrail
      Contact( "EstadosSup".Sup7_2 )
   END_RUNG wire#w1
   RUNG wire#powerrail
      Contact( "EstadosSup".Sup7_3 )
   END_RUNG wire#w1
   RUNG wire#powerrail
      Contact( "EstadosSup".Sup11_2 )
   END_RUNG wire#w1
   // the same network as SCL:
   "Des_Eventos".d_AT1_On := "EstadosSup".Sup5_1 OR "EstadosSup".Sup7_2 OR "EstadosSup".Sup7_3 OR "EstadosSup".Sup11_2;
END_REGION

REGION Network 2: Desabilita o avanço atuador 2
   RUNG wire#powerrail
      Contact( "EstadosSup".Sup6_1 )
      wire#w1
      Coil( "Des_Eventos".d_AT2_On )
   END_RUNG
   RUNG wire#powerrail
      Contact( "EstadosSup".Sup8_2 )
   END_RUNG wire#w1
   RUNG wire#powerrail
      Contact( "EstadosSup".Sup8_3 )
   END_RUNG wire#w1
   RUNG wire#powerrail
      Contact( "EstadosSup".Sup12_2 )
   END_RUNG wire#w1
   // the same network as SCL:
   "Des_Eventos".d_AT2_On := "EstadosSup".Sup6_1 OR "EstadosSup".Sup8_2 OR "EstadosSup".Sup8_3 OR "EstadosSup".Sup12_2;
END_REGION

REGION Network 3: Desabilita o ligar esteira 1
   RUNG wire#powerrail
      Contact( "EstadosSup".Sup9_2 )
      wire#w1
      Coil( "Des_Eventos".d_E1_On )
   END_RUNG
   RUNG wire#powerrail
      Contact( "EstadosSup".Sup10_2 )
   END_RUNG wire#w1
   RUNG wire#powerrail
      Contact( "EstadosSup".Sup12_2 )
   END_RUNG wire#w1
   RUNG wire#powerrail
      Contact( "EstadosSup".Sup14_2 )
   END_RUNG wire#w1
   // the same network as SCL:
   "Des_Eventos".d_E1_On := "EstadosSup".Sup9_2 OR "EstadosSup".Sup10_2 OR "EstadosSup".Sup12_2 OR "EstadosSup".Sup14_2;
END_REGION

REGION Network 4: Desabilita o desligar esteira 1
   RUNG wire#powerrail
      Contact( "EstadosSup".Sup1_2 )
      wire#w1
      Coil( "Des_Eventos".d_E1_Off )
   END_RUNG
   RUNG wire#powerrail
      Contact( "EstadosSup".Sup13_1 )
   END_RUNG wire#w1
   RUNG wire#powerrail
      Contact( "EstadosSup".Sup13_3 )
   END_RUNG wire#w1
   RUNG wire#powerrail
      Contact( "EstadosSup".Sup13_4 )
   END_RUNG wire#w1
   RUNG wire#powerrail
      Contact( "EstadosSup".Sup14_2 )
   END_RUNG wire#w1
   // the same network as SCL:
   "Des_Eventos".d_E1_Off := "EstadosSup".Sup1_2 OR "EstadosSup".Sup13_1 OR "EstadosSup".Sup13_3 OR "EstadosSup".Sup13_4 OR "EstadosSup".Sup14_2;
END_REGION

REGION Network 5: Desabilita o ligar esteira 2
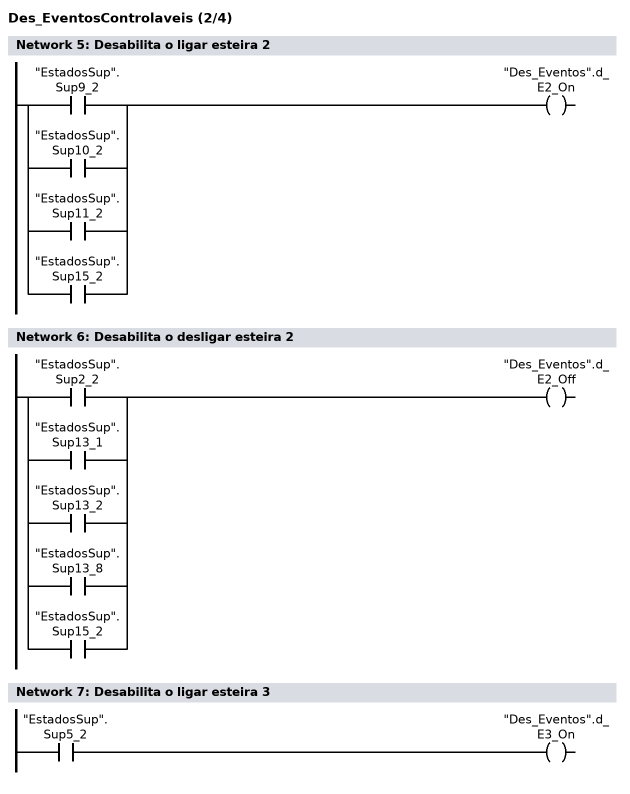
   RUNG wire#powerrail
      Contact( "EstadosSup".Sup9_2 )
      wire#w1
      Coil( "Des_Eventos".d_E2_On )
   END_RUNG
   RUNG wire#powerrail
      Contact( "EstadosSup".Sup10_2 )
   END_RUNG wire#w1
   RUNG wire#powerrail
      Contact( "EstadosSup".Sup11_2 )
   END_RUNG wire#w1
   RUNG wire#powerrail
      Contact( "EstadosSup".Sup15_2 )
   END_RUNG wire#w1
   // the same network as SCL:
   "Des_Eventos".d_E2_On := "EstadosSup".Sup9_2 OR "EstadosSup".Sup10_2 OR "EstadosSup".Sup11_2 OR "EstadosSup".Sup15_2;
END_REGION

REGION Network 6: Desabilita o desligar esteira 2
   RUNG wire#powerrail
      Contact( "EstadosSup".Sup2_2 )
      wire#w1
      Coil( "Des_Eventos".d_E2_Off )
   END_RUNG
   RUNG wire#powerrail
      Contact( "EstadosSup".Sup13_1 )
   END_RUNG wire#w1
   RUNG wire#powerrail
      Contact( "EstadosSup".Sup13_2 )
   END_RUNG wire#w1
   RUNG wire#powerrail
      Contact( "EstadosSup".Sup13_8 )
   END_RUNG wire#w1
   RUNG wire#powerrail
      Contact( "EstadosSup".Sup15_2 )
   END_RUNG wire#w1
   // the same network as SCL:
   "Des_Eventos".d_E2_Off := "EstadosSup".Sup2_2 OR "EstadosSup".Sup13_1 OR "EstadosSup".Sup13_2 OR "EstadosSup".Sup13_8 OR "EstadosSup".Sup15_2;
END_REGION

REGION Network 7: Desabilita o ligar esteira 3
   RUNG wire#powerrail
      Contact( "EstadosSup".Sup5_2 )
      Coil( "Des_Eventos".d_E3_On )
   END_RUNG
   // the same network as SCL:
   "Des_Eventos".d_E3_On := "EstadosSup".Sup5_2;
END_REGION

REGION Network 8: Desabilita o desligar esteira 3
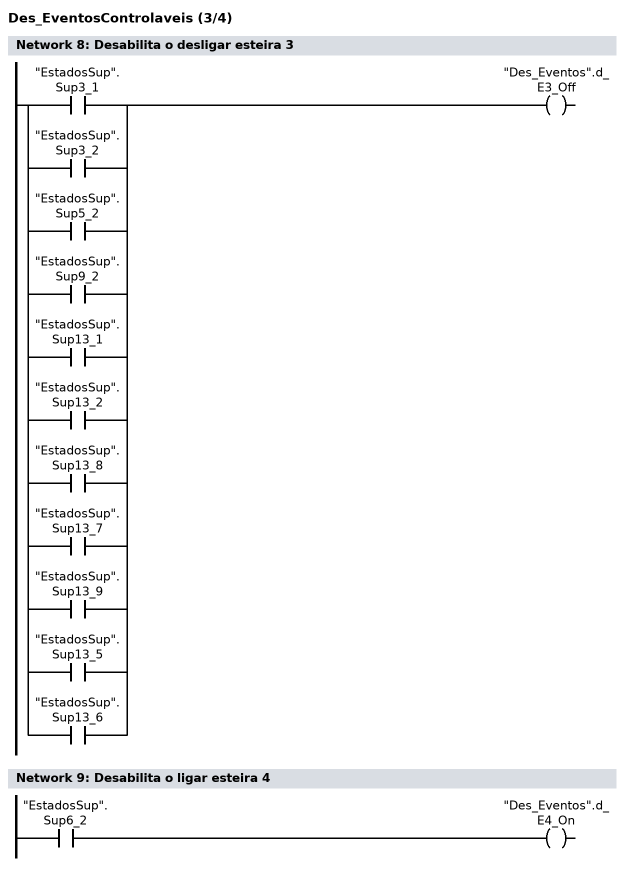
   RUNG wire#powerrail
      Contact( "EstadosSup".Sup3_1 )
      wire#w1
      Coil( "Des_Eventos".d_E3_Off )
   END_RUNG
   RUNG wire#powerrail
      Contact( "EstadosSup".Sup3_2 )
   END_RUNG wire#w1
   RUNG wire#powerrail
      Contact( "EstadosSup".Sup5_2 )
   END_RUNG wire#w1
   RUNG wire#powerrail
      Contact( "EstadosSup".Sup9_2 )
   END_RUNG wire#w1
   RUNG wire#powerrail
      Contact( "EstadosSup".Sup13_1 )
   END_RUNG wire#w1
   RUNG wire#powerrail
      Contact( "EstadosSup".Sup13_2 )
   END_RUNG wire#w1
   RUNG wire#powerrail
      Contact( "EstadosSup".Sup13_8 )
   END_RUNG wire#w1
   RUNG wire#powerrail
      Contact( "EstadosSup".Sup13_7 )
   END_RUNG wire#w1
   RUNG wire#powerrail
      Contact( "EstadosSup".Sup13_9 )
   END_RUNG wire#w1
   RUNG wire#powerrail
      Contact( "EstadosSup".Sup13_5 )
   END_RUNG wire#w1
   RUNG wire#powerrail
      Contact( "EstadosSup".Sup13_6 )
   END_RUNG wire#w1
   // the same network as SCL:
   "Des_Eventos".d_E3_Off := "EstadosSup".Sup3_1 OR "EstadosSup".Sup3_2 OR "EstadosSup".Sup5_2 OR "EstadosSup".Sup9_2 OR "EstadosSup".Sup13_1 OR "EstadosSup".Sup13_2 OR "EstadosSup".Sup13_8 OR "EstadosSup".Sup13_7 OR "EstadosSup".Sup13_9 OR "EstadosSup".Sup13_5 OR "EstadosSup".Sup13_6;
END_REGION

REGION Network 9: Desabilita o ligar esteira 4
   RUNG wire#powerrail
      Contact( "EstadosSup".Sup6_2 )
      Coil( "Des_Eventos".d_E4_On )
   END_RUNG
   // the same network as SCL:
   "Des_Eventos".d_E4_On := "EstadosSup".Sup6_2;
END_REGION

REGION Network 10: Desabilita o desligar esteira 4
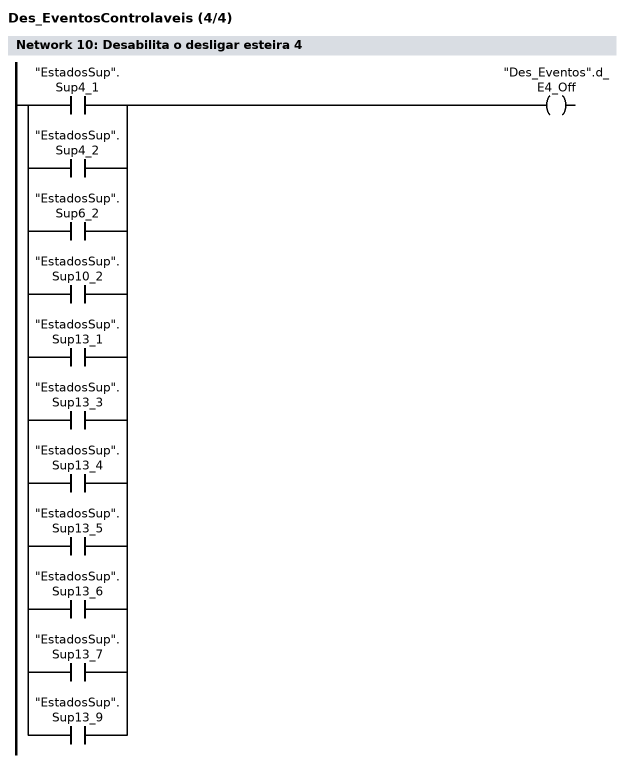
   RUNG wire#powerrail
      Contact( "EstadosSup".Sup4_1 )
      wire#w1
      Coil( "Des_Eventos".d_E4_Off )
   END_RUNG
   RUNG wire#powerrail
      Contact( "EstadosSup".Sup4_2 )
   END_RUNG wire#w1
   RUNG wire#powerrail
      Contact( "EstadosSup".Sup6_2 )
   END_RUNG wire#w1
   RUNG wire#powerrail
      Contact( "EstadosSup".Sup10_2 )
   END_RUNG wire#w1
   RUNG wire#powerrail
      Contact( "EstadosSup".Sup13_1 )
   END_RUNG wire#w1
   RUNG wire#powerrail
      Contact( "EstadosSup".Sup13_3 )
   END_RUNG wire#w1
   RUNG wire#powerrail
      Contact( "EstadosSup".Sup13_4 )
   END_RUNG wire#w1
   RUNG wire#powerrail
      Contact( "EstadosSup".Sup13_5 )
   END_RUNG wire#w1
   RUNG wire#powerrail
      Contact( "EstadosSup".Sup13_6 )
   END_RUNG wire#w1
   RUNG wire#powerrail
      Contact( "EstadosSup".Sup13_7 )
   END_RUNG wire#w1
   RUNG wire#powerrail
      Contact( "EstadosSup".Sup13_9 )
   END_RUNG wire#w1
   // the same network as SCL:
   "Des_Eventos".d_E4_Off := "EstadosSup".Sup4_1 OR "EstadosSup".Sup4_2 OR "EstadosSup".Sup6_2 OR "EstadosSup".Sup10_2 OR "EstadosSup".Sup13_1 OR "EstadosSup".Sup13_3 OR "EstadosSup".Sup13_4 OR "EstadosSup".Sup13_5 OR "EstadosSup".Sup13_6 OR "EstadosSup".Sup13_7 OR "EstadosSup".Sup13_9;
END_REGION
END_FUNCTION

FUNCTION "Ger_Eventos_Contr" : Void   // FC6, LAD
TITLE = Geração de eventos controláveis e atualização dos modelos do SP.
{ S7_Optimized_Access := 'TRUE' }
VERSION : 0.1
   VAR_TEMP   // added for the SCL form of the ladder/FBD networks
      _w1 : Bool;
   END_VAR
BEGIN

REGION Network 1: Geração evento de acionar atuador 1
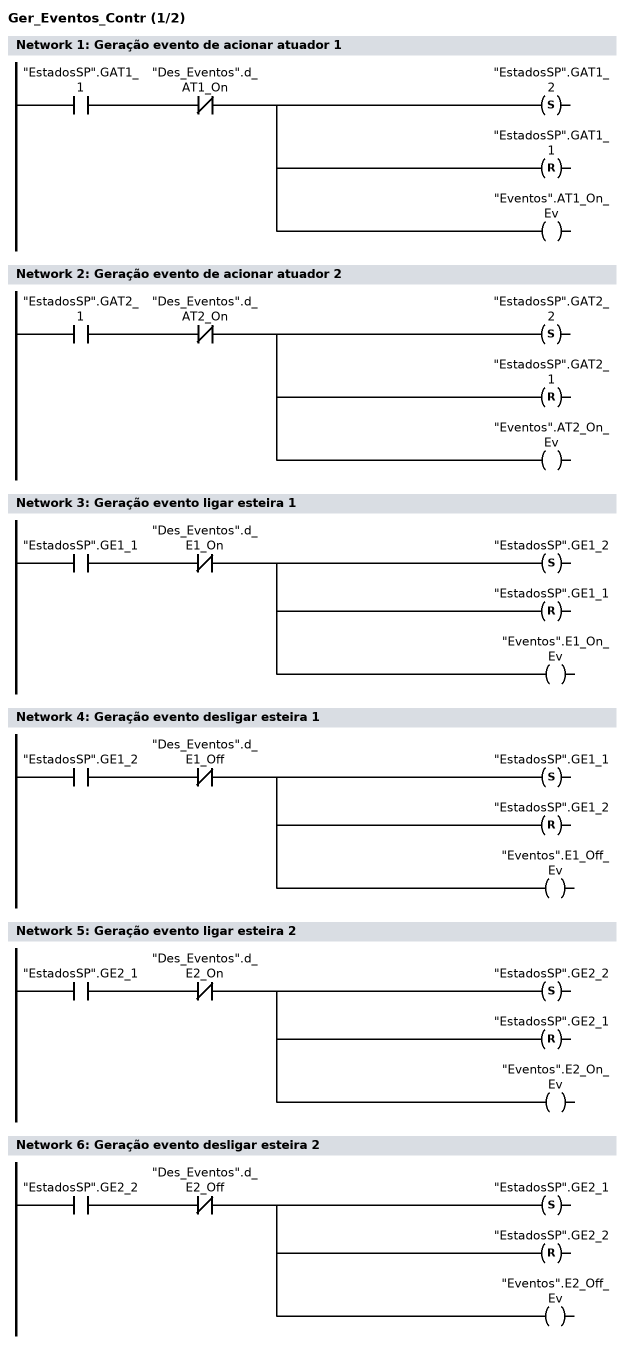
   RUNG wire#powerrail
      Contact( "EstadosSP".GAT1_1 )
      I_Contact( "Des_Eventos".d_AT1_On )
      wire#w1
      S_Coil( "EstadosSP".GAT1_2 )
   END_RUNG
   RUNG wire#w1
      R_Coil( "EstadosSP".GAT1_1 )
   END_RUNG
   RUNG wire#w1
      Coil( "Eventos".AT1_On_Ev )
   END_RUNG
   // the same network as SCL:
   #_w1 := "EstadosSP".GAT1_1 AND NOT "Des_Eventos".d_AT1_On;
   IF #_w1 THEN
       "EstadosSP".GAT1_2 := TRUE;
       "EstadosSP".GAT1_1 := FALSE;
   END_IF;
   "Eventos".AT1_On_Ev := #_w1;
END_REGION

REGION Network 2: Geração evento de acionar atuador 2
   RUNG wire#powerrail
      Contact( "EstadosSP".GAT2_1 )
      I_Contact( "Des_Eventos".d_AT2_On )
      wire#w1
      S_Coil( "EstadosSP".GAT2_2 )
   END_RUNG
   RUNG wire#w1
      R_Coil( "EstadosSP".GAT2_1 )
   END_RUNG
   RUNG wire#w1
      Coil( "Eventos".AT2_On_Ev )
   END_RUNG
   // the same network as SCL:
   #_w1 := "EstadosSP".GAT2_1 AND NOT "Des_Eventos".d_AT2_On;
   IF #_w1 THEN
       "EstadosSP".GAT2_2 := TRUE;
       "EstadosSP".GAT2_1 := FALSE;
   END_IF;
   "Eventos".AT2_On_Ev := #_w1;
END_REGION

REGION Network 3: Geração evento ligar esteira 1
   RUNG wire#powerrail
      Contact( "EstadosSP".GE1_1 )
      I_Contact( "Des_Eventos".d_E1_On )
      wire#w1
      S_Coil( "EstadosSP".GE1_2 )
   END_RUNG
   RUNG wire#w1
      R_Coil( "EstadosSP".GE1_1 )
   END_RUNG
   RUNG wire#w1
      Coil( "Eventos".E1_On_Ev )
   END_RUNG
   // the same network as SCL:
   #_w1 := "EstadosSP".GE1_1 AND NOT "Des_Eventos".d_E1_On;
   IF #_w1 THEN
       "EstadosSP".GE1_2 := TRUE;
       "EstadosSP".GE1_1 := FALSE;
   END_IF;
   "Eventos".E1_On_Ev := #_w1;
END_REGION

REGION Network 4: Geração evento desligar esteira 1
   RUNG wire#powerrail
      Contact( "EstadosSP".GE1_2 )
      I_Contact( "Des_Eventos".d_E1_Off )
      wire#w1
      S_Coil( "EstadosSP".GE1_1 )
   END_RUNG
   RUNG wire#w1
      R_Coil( "EstadosSP".GE1_2 )
   END_RUNG
   RUNG wire#w1
      Coil( "Eventos".E1_Off_Ev )
   END_RUNG
   // the same network as SCL:
   #_w1 := "EstadosSP".GE1_2 AND NOT "Des_Eventos".d_E1_Off;
   IF #_w1 THEN
       "EstadosSP".GE1_1 := TRUE;
       "EstadosSP".GE1_2 := FALSE;
   END_IF;
   "Eventos".E1_Off_Ev := #_w1;
END_REGION

REGION Network 5: Geração evento ligar esteira 2
   RUNG wire#powerrail
      Contact( "EstadosSP".GE2_1 )
      I_Contact( "Des_Eventos".d_E2_On )
      wire#w1
      S_Coil( "EstadosSP".GE2_2 )
   END_RUNG
   RUNG wire#w1
      R_Coil( "EstadosSP".GE2_1 )
   END_RUNG
   RUNG wire#w1
      Coil( "Eventos".E2_On_Ev )
   END_RUNG
   // the same network as SCL:
   #_w1 := "EstadosSP".GE2_1 AND NOT "Des_Eventos".d_E2_On;
   IF #_w1 THEN
       "EstadosSP".GE2_2 := TRUE;
       "EstadosSP".GE2_1 := FALSE;
   END_IF;
   "Eventos".E2_On_Ev := #_w1;
END_REGION

REGION Network 6: Geração evento desligar esteira 2
   RUNG wire#powerrail
      Contact( "EstadosSP".GE2_2 )
      I_Contact( "Des_Eventos".d_E2_Off )
      wire#w1
      S_Coil( "EstadosSP".GE2_1 )
   END_RUNG
   RUNG wire#w1
      R_Coil( "EstadosSP".GE2_2 )
   END_RUNG
   RUNG wire#w1
      Coil( "Eventos".E2_Off_Ev )
   END_RUNG
   // the same network as SCL:
   #_w1 := "EstadosSP".GE2_2 AND NOT "Des_Eventos".d_E2_Off;
   IF #_w1 THEN
       "EstadosSP".GE2_1 := TRUE;
       "EstadosSP".GE2_2 := FALSE;
   END_IF;
   "Eventos".E2_Off_Ev := #_w1;
END_REGION

REGION Network 7: Geração evento ligar esteira 3
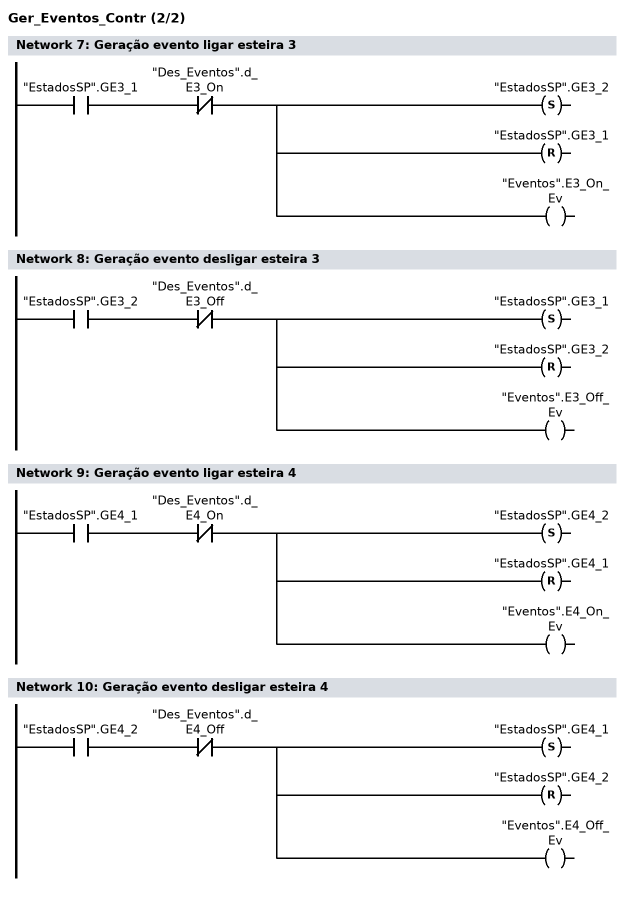
   RUNG wire#powerrail
      Contact( "EstadosSP".GE3_1 )
      I_Contact( "Des_Eventos".d_E3_On )
      wire#w1
      S_Coil( "EstadosSP".GE3_2 )
   END_RUNG
   RUNG wire#w1
      R_Coil( "EstadosSP".GE3_1 )
   END_RUNG
   RUNG wire#w1
      Coil( "Eventos".E3_On_Ev )
   END_RUNG
   // the same network as SCL:
   #_w1 := "EstadosSP".GE3_1 AND NOT "Des_Eventos".d_E3_On;
   IF #_w1 THEN
       "EstadosSP".GE3_2 := TRUE;
       "EstadosSP".GE3_1 := FALSE;
   END_IF;
   "Eventos".E3_On_Ev := #_w1;
END_REGION

REGION Network 8: Geração evento desligar esteira 3
   RUNG wire#powerrail
      Contact( "EstadosSP".GE3_2 )
      I_Contact( "Des_Eventos".d_E3_Off )
      wire#w1
      S_Coil( "EstadosSP".GE3_1 )
   END_RUNG
   RUNG wire#w1
      R_Coil( "EstadosSP".GE3_2 )
   END_RUNG
   RUNG wire#w1
      Coil( "Eventos".E3_Off_Ev )
   END_RUNG
   // the same network as SCL:
   #_w1 := "EstadosSP".GE3_2 AND NOT "Des_Eventos".d_E3_Off;
   IF #_w1 THEN
       "EstadosSP".GE3_1 := TRUE;
       "EstadosSP".GE3_2 := FALSE;
   END_IF;
   "Eventos".E3_Off_Ev := #_w1;
END_REGION

REGION Network 9: Geração evento ligar esteira 4
   RUNG wire#powerrail
      Contact( "EstadosSP".GE4_1 )
      I_Contact( "Des_Eventos".d_E4_On )
      wire#w1
      S_Coil( "EstadosSP".GE4_2 )
   END_RUNG
   RUNG wire#w1
      R_Coil( "EstadosSP".GE4_1 )
   END_RUNG
   RUNG wire#w1
      Coil( "Eventos".E4_On_Ev )
   END_RUNG
   // the same network as SCL:
   #_w1 := "EstadosSP".GE4_1 AND NOT "Des_Eventos".d_E4_On;
   IF #_w1 THEN
       "EstadosSP".GE4_2 := TRUE;
       "EstadosSP".GE4_1 := FALSE;
   END_IF;
   "Eventos".E4_On_Ev := #_w1;
END_REGION

REGION Network 10: Geração evento desligar esteira 4
   RUNG wire#powerrail
      Contact( "EstadosSP".GE4_2 )
      I_Contact( "Des_Eventos".d_E4_Off )
      wire#w1
      S_Coil( "EstadosSP".GE4_1 )
   END_RUNG
   RUNG wire#w1
      R_Coil( "EstadosSP".GE4_2 )
   END_RUNG
   RUNG wire#w1
      Coil( "Eventos".E4_Off_Ev )
   END_RUNG
   // the same network as SCL:
   #_w1 := "EstadosSP".GE4_2 AND NOT "Des_Eventos".d_E4_Off;
   IF #_w1 THEN
       "EstadosSP".GE4_1 := TRUE;
       "EstadosSP".GE4_2 := FALSE;
   END_IF;
   "Eventos".E4_Off_Ev := #_w1;
END_REGION
END_FUNCTION

FUNCTION "At_Sup_Controlaveis" : Void   // FC7, LAD
TITLE = Atualização dos estados dos supervisores reduzidos, devido a eventos controláveis
{ S7_Optimized_Access := 'TRUE' }
VERSION : 0.1
BEGIN

REGION Network 1: Atualização do supervisor 3, estado 3 para estado 1.
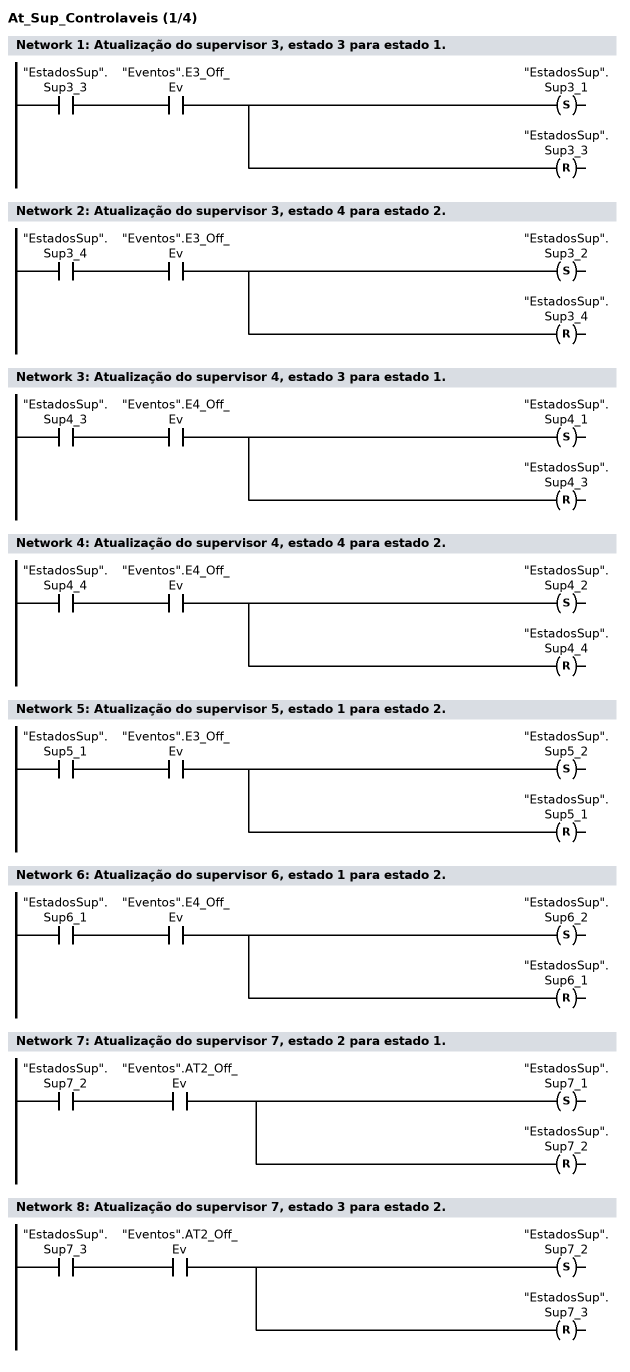
   RUNG wire#powerrail
      Contact( "EstadosSup".Sup3_3 )
      Contact( "Eventos".E3_Off_Ev )
      wire#w1
      S_Coil( "EstadosSup".Sup3_1 )
   END_RUNG
   RUNG wire#w1
      R_Coil( "EstadosSup".Sup3_3 )
   END_RUNG
   // the same network as SCL:
   IF "EstadosSup".Sup3_3 AND "Eventos".E3_Off_Ev THEN
       "EstadosSup".Sup3_1 := TRUE;
       "EstadosSup".Sup3_3 := FALSE;
   END_IF;
END_REGION

REGION Network 2: Atualização do supervisor 3, estado 4 para estado 2.
   RUNG wire#powerrail
      Contact( "EstadosSup".Sup3_4 )
      Contact( "Eventos".E3_Off_Ev )
      wire#w1
      S_Coil( "EstadosSup".Sup3_2 )
   END_RUNG
   RUNG wire#w1
      R_Coil( "EstadosSup".Sup3_4 )
   END_RUNG
   // the same network as SCL:
   IF "EstadosSup".Sup3_4 AND "Eventos".E3_Off_Ev THEN
       "EstadosSup".Sup3_2 := TRUE;
       "EstadosSup".Sup3_4 := FALSE;
   END_IF;
END_REGION

REGION Network 3: Atualização do supervisor 4, estado 3 para estado 1.
   RUNG wire#powerrail
      Contact( "EstadosSup".Sup4_3 )
      Contact( "Eventos".E4_Off_Ev )
      wire#w1
      S_Coil( "EstadosSup".Sup4_1 )
   END_RUNG
   RUNG wire#w1
      R_Coil( "EstadosSup".Sup4_3 )
   END_RUNG
   // the same network as SCL:
   IF "EstadosSup".Sup4_3 AND "Eventos".E4_Off_Ev THEN
       "EstadosSup".Sup4_1 := TRUE;
       "EstadosSup".Sup4_3 := FALSE;
   END_IF;
END_REGION

REGION Network 4: Atualização do supervisor 4, estado 4 para estado 2.
   RUNG wire#powerrail
      Contact( "EstadosSup".Sup4_4 )
      Contact( "Eventos".E4_Off_Ev )
      wire#w1
      S_Coil( "EstadosSup".Sup4_2 )
   END_RUNG
   RUNG wire#w1
      R_Coil( "EstadosSup".Sup4_4 )
   END_RUNG
   // the same network as SCL:
   IF "EstadosSup".Sup4_4 AND "Eventos".E4_Off_Ev THEN
       "EstadosSup".Sup4_2 := TRUE;
       "EstadosSup".Sup4_4 := FALSE;
   END_IF;
END_REGION

REGION Network 5: Atualização do supervisor 5, estado 1 para estado 2.
   RUNG wire#powerrail
      Contact( "EstadosSup".Sup5_1 )
      Contact( "Eventos".E3_Off_Ev )
      wire#w1
      S_Coil( "EstadosSup".Sup5_2 )
   END_RUNG
   RUNG wire#w1
      R_Coil( "EstadosSup".Sup5_1 )
   END_RUNG
   // the same network as SCL:
   IF "EstadosSup".Sup5_1 AND "Eventos".E3_Off_Ev THEN
       "EstadosSup".Sup5_2 := TRUE;
       "EstadosSup".Sup5_1 := FALSE;
   END_IF;
END_REGION

REGION Network 6: Atualização do supervisor 6, estado 1 para estado 2.
   RUNG wire#powerrail
      Contact( "EstadosSup".Sup6_1 )
      Contact( "Eventos".E4_Off_Ev )
      wire#w1
      S_Coil( "EstadosSup".Sup6_2 )
   END_RUNG
   RUNG wire#w1
      R_Coil( "EstadosSup".Sup6_1 )
   END_RUNG
   // the same network as SCL:
   IF "EstadosSup".Sup6_1 AND "Eventos".E4_Off_Ev THEN
       "EstadosSup".Sup6_2 := TRUE;
       "EstadosSup".Sup6_1 := FALSE;
   END_IF;
END_REGION

REGION Network 7: Atualização do supervisor 7, estado 2 para estado 1.
   RUNG wire#powerrail
      Contact( "EstadosSup".Sup7_2 )
      Contact( "Eventos".AT2_Off_Ev )
      wire#w1
      S_Coil( "EstadosSup".Sup7_1 )
   END_RUNG
   RUNG wire#w1
      R_Coil( "EstadosSup".Sup7_2 )
   END_RUNG
   // the same network as SCL:
   IF "EstadosSup".Sup7_2 AND "Eventos".AT2_Off_Ev THEN
       "EstadosSup".Sup7_1 := TRUE;
       "EstadosSup".Sup7_2 := FALSE;
   END_IF;
END_REGION

REGION Network 8: Atualização do supervisor 7, estado 3 para estado 2.
   RUNG wire#powerrail
      Contact( "EstadosSup".Sup7_3 )
      Contact( "Eventos".AT2_Off_Ev )
      wire#w1
      S_Coil( "EstadosSup".Sup7_2 )
   END_RUNG
   RUNG wire#w1
      R_Coil( "EstadosSup".Sup7_3 )
   END_RUNG
   // the same network as SCL:
   IF "EstadosSup".Sup7_3 AND "Eventos".AT2_Off_Ev THEN
       "EstadosSup".Sup7_2 := TRUE;
       "EstadosSup".Sup7_3 := FALSE;
   END_IF;
END_REGION

REGION Network 9: Atualização do supervisor 8, estado 2 para estado 1.
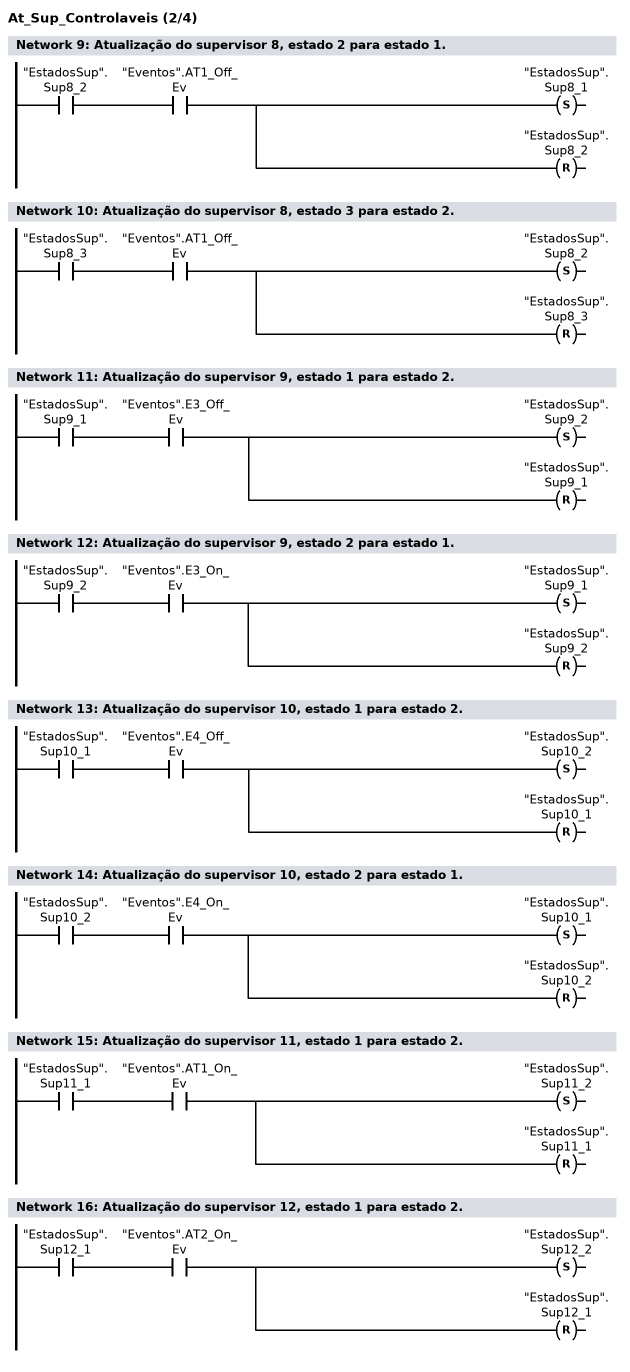
   RUNG wire#powerrail
      Contact( "EstadosSup".Sup8_2 )
      Contact( "Eventos".AT1_Off_Ev )
      wire#w1
      S_Coil( "EstadosSup".Sup8_1 )
   END_RUNG
   RUNG wire#w1
      R_Coil( "EstadosSup".Sup8_2 )
   END_RUNG
   // the same network as SCL:
   IF "EstadosSup".Sup8_2 AND "Eventos".AT1_Off_Ev THEN
       "EstadosSup".Sup8_1 := TRUE;
       "EstadosSup".Sup8_2 := FALSE;
   END_IF;
END_REGION

REGION Network 10: Atualização do supervisor 8, estado 3 para estado 2.
   RUNG wire#powerrail
      Contact( "EstadosSup".Sup8_3 )
      Contact( "Eventos".AT1_Off_Ev )
      wire#w1
      S_Coil( "EstadosSup".Sup8_2 )
   END_RUNG
   RUNG wire#w1
      R_Coil( "EstadosSup".Sup8_3 )
   END_RUNG
   // the same network as SCL:
   IF "EstadosSup".Sup8_3 AND "Eventos".AT1_Off_Ev THEN
       "EstadosSup".Sup8_2 := TRUE;
       "EstadosSup".Sup8_3 := FALSE;
   END_IF;
END_REGION

REGION Network 11: Atualização do supervisor 9, estado 1 para estado 2.
   RUNG wire#powerrail
      Contact( "EstadosSup".Sup9_1 )
      Contact( "Eventos".E3_Off_Ev )
      wire#w1
      S_Coil( "EstadosSup".Sup9_2 )
   END_RUNG
   RUNG wire#w1
      R_Coil( "EstadosSup".Sup9_1 )
   END_RUNG
   // the same network as SCL:
   IF "EstadosSup".Sup9_1 AND "Eventos".E3_Off_Ev THEN
       "EstadosSup".Sup9_2 := TRUE;
       "EstadosSup".Sup9_1 := FALSE;
   END_IF;
END_REGION

REGION Network 12: Atualização do supervisor 9, estado 2 para estado 1.
   RUNG wire#powerrail
      Contact( "EstadosSup".Sup9_2 )
      Contact( "Eventos".E3_On_Ev )
      wire#w1
      S_Coil( "EstadosSup".Sup9_1 )
   END_RUNG
   RUNG wire#w1
      R_Coil( "EstadosSup".Sup9_2 )
   END_RUNG
   // the same network as SCL:
   IF "EstadosSup".Sup9_2 AND "Eventos".E3_On_Ev THEN
       "EstadosSup".Sup9_1 := TRUE;
       "EstadosSup".Sup9_2 := FALSE;
   END_IF;
END_REGION

REGION Network 13: Atualização do supervisor 10, estado 1 para estado 2.
   RUNG wire#powerrail
      Contact( "EstadosSup".Sup10_1 )
      Contact( "Eventos".E4_Off_Ev )
      wire#w1
      S_Coil( "EstadosSup".Sup10_2 )
   END_RUNG
   RUNG wire#w1
      R_Coil( "EstadosSup".Sup10_1 )
   END_RUNG
   // the same network as SCL:
   IF "EstadosSup".Sup10_1 AND "Eventos".E4_Off_Ev THEN
       "EstadosSup".Sup10_2 := TRUE;
       "EstadosSup".Sup10_1 := FALSE;
   END_IF;
END_REGION

REGION Network 14: Atualização do supervisor 10, estado 2 para estado 1.
   RUNG wire#powerrail
      Contact( "EstadosSup".Sup10_2 )
      Contact( "Eventos".E4_On_Ev )
      wire#w1
      S_Coil( "EstadosSup".Sup10_1 )
   END_RUNG
   RUNG wire#w1
      R_Coil( "EstadosSup".Sup10_2 )
   END_RUNG
   // the same network as SCL:
   IF "EstadosSup".Sup10_2 AND "Eventos".E4_On_Ev THEN
       "EstadosSup".Sup10_1 := TRUE;
       "EstadosSup".Sup10_2 := FALSE;
   END_IF;
END_REGION

REGION Network 15: Atualização do supervisor 11, estado 1 para estado 2.
   RUNG wire#powerrail
      Contact( "EstadosSup".Sup11_1 )
      Contact( "Eventos".AT1_On_Ev )
      wire#w1
      S_Coil( "EstadosSup".Sup11_2 )
   END_RUNG
   RUNG wire#w1
      R_Coil( "EstadosSup".Sup11_1 )
   END_RUNG
   // the same network as SCL:
   IF "EstadosSup".Sup11_1 AND "Eventos".AT1_On_Ev THEN
       "EstadosSup".Sup11_2 := TRUE;
       "EstadosSup".Sup11_1 := FALSE;
   END_IF;
END_REGION

REGION Network 16: Atualização do supervisor 12, estado 1 para estado 2.
   RUNG wire#powerrail
      Contact( "EstadosSup".Sup12_1 )
      Contact( "Eventos".AT2_On_Ev )
      wire#w1
      S_Coil( "EstadosSup".Sup12_2 )
   END_RUNG
   RUNG wire#w1
      R_Coil( "EstadosSup".Sup12_1 )
   END_RUNG
   // the same network as SCL:
   IF "EstadosSup".Sup12_1 AND "Eventos".AT2_On_Ev THEN
       "EstadosSup".Sup12_2 := TRUE;
       "EstadosSup".Sup12_1 := FALSE;
   END_IF;
END_REGION

REGION Network 17: Atualização do supervisor 13, estado 2 para estado 7.
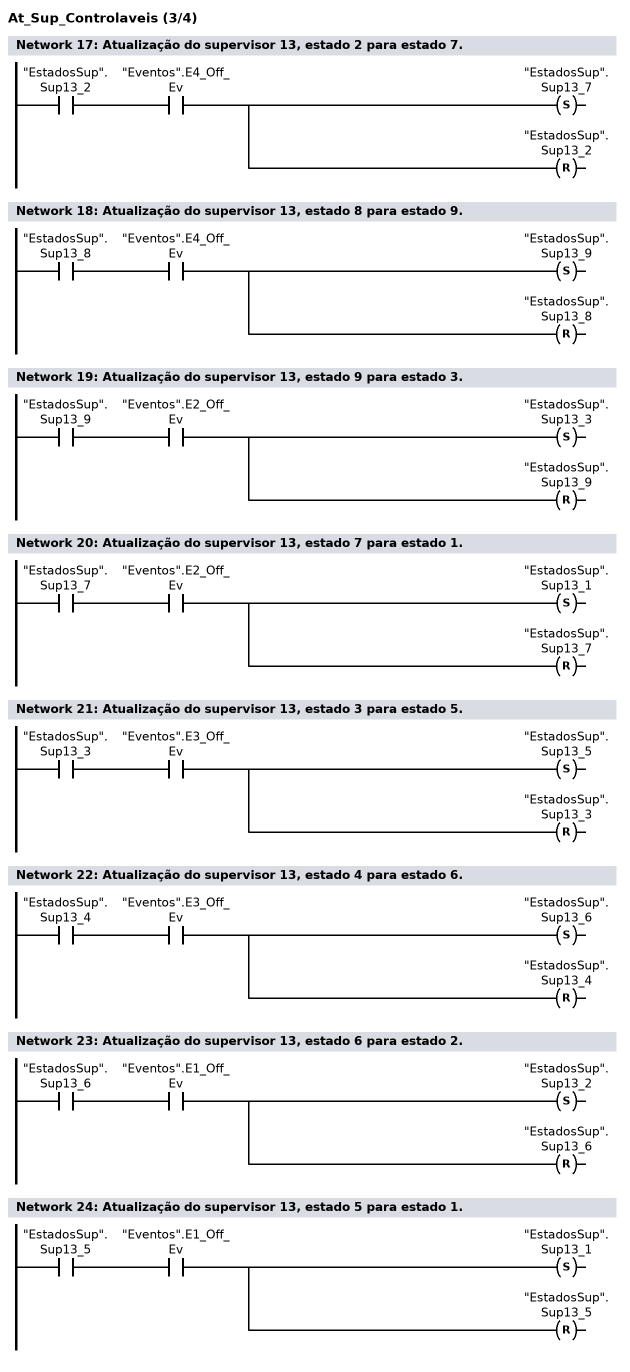
   RUNG wire#powerrail
      Contact( "EstadosSup".Sup13_2 )
      Contact( "Eventos".E4_Off_Ev )
      wire#w1
      S_Coil( "EstadosSup".Sup13_7 )
   END_RUNG
   RUNG wire#w1
      R_Coil( "EstadosSup".Sup13_2 )
   END_RUNG
   // the same network as SCL:
   IF "EstadosSup".Sup13_2 AND "Eventos".E4_Off_Ev THEN
       "EstadosSup".Sup13_7 := TRUE;
       "EstadosSup".Sup13_2 := FALSE;
   END_IF;
END_REGION

REGION Network 18: Atualização do supervisor 13, estado 8 para estado 9.
   RUNG wire#powerrail
      Contact( "EstadosSup".Sup13_8 )
      Contact( "Eventos".E4_Off_Ev )
      wire#w1
      S_Coil( "EstadosSup".Sup13_9 )
   END_RUNG
   RUNG wire#w1
      R_Coil( "EstadosSup".Sup13_8 )
   END_RUNG
   // the same network as SCL:
   IF "EstadosSup".Sup13_8 AND "Eventos".E4_Off_Ev THEN
       "EstadosSup".Sup13_9 := TRUE;
       "EstadosSup".Sup13_8 := FALSE;
   END_IF;
END_REGION

REGION Network 19: Atualização do supervisor 13, estado 9 para estado 3.
   RUNG wire#powerrail
      Contact( "EstadosSup".Sup13_9 )
      Contact( "Eventos".E2_Off_Ev )
      wire#w1
      S_Coil( "EstadosSup".Sup13_3 )
   END_RUNG
   RUNG wire#w1
      R_Coil( "EstadosSup".Sup13_9 )
   END_RUNG
   // the same network as SCL:
   IF "EstadosSup".Sup13_9 AND "Eventos".E2_Off_Ev THEN
       "EstadosSup".Sup13_3 := TRUE;
       "EstadosSup".Sup13_9 := FALSE;
   END_IF;
END_REGION

REGION Network 20: Atualização do supervisor 13, estado 7 para estado 1.
   RUNG wire#powerrail
      Contact( "EstadosSup".Sup13_7 )
      Contact( "Eventos".E2_Off_Ev )
      wire#w1
      S_Coil( "EstadosSup".Sup13_1 )
   END_RUNG
   RUNG wire#w1
      R_Coil( "EstadosSup".Sup13_7 )
   END_RUNG
   // the same network as SCL:
   IF "EstadosSup".Sup13_7 AND "Eventos".E2_Off_Ev THEN
       "EstadosSup".Sup13_1 := TRUE;
       "EstadosSup".Sup13_7 := FALSE;
   END_IF;
END_REGION

REGION Network 21: Atualização do supervisor 13, estado 3 para estado 5.
   RUNG wire#powerrail
      Contact( "EstadosSup".Sup13_3 )
      Contact( "Eventos".E3_Off_Ev )
      wire#w1
      S_Coil( "EstadosSup".Sup13_5 )
   END_RUNG
   RUNG wire#w1
      R_Coil( "EstadosSup".Sup13_3 )
   END_RUNG
   // the same network as SCL:
   IF "EstadosSup".Sup13_3 AND "Eventos".E3_Off_Ev THEN
       "EstadosSup".Sup13_5 := TRUE;
       "EstadosSup".Sup13_3 := FALSE;
   END_IF;
END_REGION

REGION Network 22: Atualização do supervisor 13, estado 4 para estado 6.
   RUNG wire#powerrail
      Contact( "EstadosSup".Sup13_4 )
      Contact( "Eventos".E3_Off_Ev )
      wire#w1
      S_Coil( "EstadosSup".Sup13_6 )
   END_RUNG
   RUNG wire#w1
      R_Coil( "EstadosSup".Sup13_4 )
   END_RUNG
   // the same network as SCL:
   IF "EstadosSup".Sup13_4 AND "Eventos".E3_Off_Ev THEN
       "EstadosSup".Sup13_6 := TRUE;
       "EstadosSup".Sup13_4 := FALSE;
   END_IF;
END_REGION

REGION Network 23: Atualização do supervisor 13, estado 6 para estado 2.
   RUNG wire#powerrail
      Contact( "EstadosSup".Sup13_6 )
      Contact( "Eventos".E1_Off_Ev )
      wire#w1
      S_Coil( "EstadosSup".Sup13_2 )
   END_RUNG
   RUNG wire#w1
      R_Coil( "EstadosSup".Sup13_6 )
   END_RUNG
   // the same network as SCL:
   IF "EstadosSup".Sup13_6 AND "Eventos".E1_Off_Ev THEN
       "EstadosSup".Sup13_2 := TRUE;
       "EstadosSup".Sup13_6 := FALSE;
   END_IF;
END_REGION

REGION Network 24: Atualização do supervisor 13, estado 5 para estado 1.
   RUNG wire#powerrail
      Contact( "EstadosSup".Sup13_5 )
      Contact( "Eventos".E1_Off_Ev )
      wire#w1
      S_Coil( "EstadosSup".Sup13_1 )
   END_RUNG
   RUNG wire#w1
      R_Coil( "EstadosSup".Sup13_5 )
   END_RUNG
   // the same network as SCL:
   IF "EstadosSup".Sup13_5 AND "Eventos".E1_Off_Ev THEN
       "EstadosSup".Sup13_1 := TRUE;
       "EstadosSup".Sup13_5 := FALSE;
   END_IF;
END_REGION

REGION Network 25: Atualização do supervisor 14, estado 1 para estado 2.
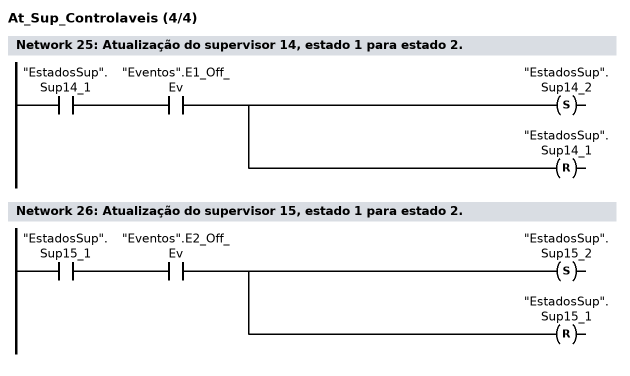
   RUNG wire#powerrail
      Contact( "EstadosSup".Sup14_1 )
      Contact( "Eventos".E1_Off_Ev )
      wire#w1
      S_Coil( "EstadosSup".Sup14_2 )
   END_RUNG
   RUNG wire#w1
      R_Coil( "EstadosSup".Sup14_1 )
   END_RUNG
   // the same network as SCL:
   IF "EstadosSup".Sup14_1 AND "Eventos".E1_Off_Ev THEN
       "EstadosSup".Sup14_2 := TRUE;
       "EstadosSup".Sup14_1 := FALSE;
   END_IF;
END_REGION

REGION Network 26: Atualização do supervisor 15, estado 1 para estado 2.
   RUNG wire#powerrail
      Contact( "EstadosSup".Sup15_1 )
      Contact( "Eventos".E2_Off_Ev )
      wire#w1
      S_Coil( "EstadosSup".Sup15_2 )
   END_RUNG
   RUNG wire#w1
      R_Coil( "EstadosSup".Sup15_1 )
   END_RUNG
   // the same network as SCL:
   IF "EstadosSup".Sup15_1 AND "Eventos".E2_Off_Ev THEN
       "EstadosSup".Sup15_2 := TRUE;
       "EstadosSup".Sup15_1 := FALSE;
   END_IF;
END_REGION
END_FUNCTION

FUNCTION "EscritaSaidas" : Void   // FC8, LAD
TITLE = Escrita nos bits de saída
{ S7_Optimized_Access := 'TRUE' }
VERSION : 0.1
BEGIN

REGION Network 1: Atuador 1
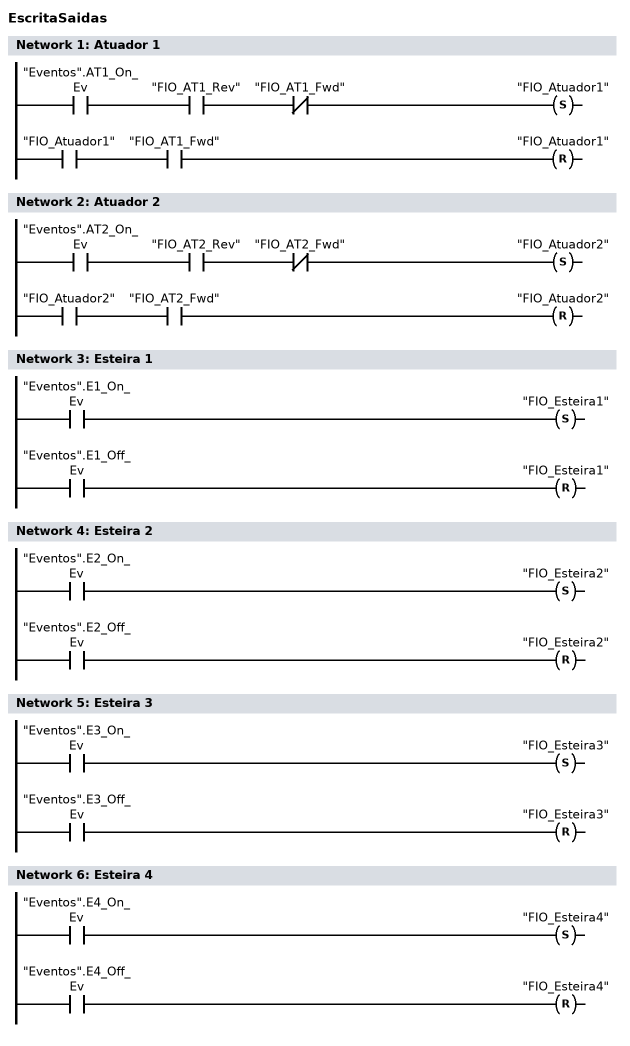
   RUNG wire#powerrail
      Contact( "Eventos".AT1_On_Ev )
      Contact( "FIO_AT1_Rev" )
      I_Contact( "FIO_AT1_Fwd" )
      S_Coil( "FIO_Atuador1" )
   END_RUNG
   RUNG wire#powerrail
      Contact( "FIO_Atuador1" )
      Contact( "FIO_AT1_Fwd" )
      R_Coil( "FIO_Atuador1" )
   END_RUNG
   // the same network as SCL:
   IF "Eventos".AT1_On_Ev AND "FIO_AT1_Rev" AND NOT "FIO_AT1_Fwd" THEN "FIO_Atuador1" := TRUE; END_IF;
   IF "FIO_Atuador1" AND "FIO_AT1_Fwd" THEN "FIO_Atuador1" := FALSE; END_IF;
END_REGION

REGION Network 2: Atuador 2
   RUNG wire#powerrail
      Contact( "Eventos".AT2_On_Ev )
      Contact( "FIO_AT2_Rev" )
      I_Contact( "FIO_AT2_Fwd" )
      S_Coil( "FIO_Atuador2" )
   END_RUNG
   RUNG wire#powerrail
      Contact( "FIO_Atuador2" )
      Contact( "FIO_AT2_Fwd" )
      R_Coil( "FIO_Atuador2" )
   END_RUNG
   // the same network as SCL:
   IF "Eventos".AT2_On_Ev AND "FIO_AT2_Rev" AND NOT "FIO_AT2_Fwd" THEN "FIO_Atuador2" := TRUE; END_IF;
   IF "FIO_Atuador2" AND "FIO_AT2_Fwd" THEN "FIO_Atuador2" := FALSE; END_IF;
END_REGION

REGION Network 3: Esteira 1
   RUNG wire#powerrail
      Contact( "Eventos".E1_On_Ev )
      S_Coil( "FIO_Esteira1" )
   END_RUNG
   RUNG wire#powerrail
      Contact( "Eventos".E1_Off_Ev )
      R_Coil( "FIO_Esteira1" )
   END_RUNG
   // the same network as SCL:
   IF "Eventos".E1_On_Ev THEN "FIO_Esteira1" := TRUE; END_IF;
   IF "Eventos".E1_Off_Ev THEN "FIO_Esteira1" := FALSE; END_IF;
END_REGION

REGION Network 4: Esteira 2
   RUNG wire#powerrail
      Contact( "Eventos".E2_On_Ev )
      S_Coil( "FIO_Esteira2" )
   END_RUNG
   RUNG wire#powerrail
      Contact( "Eventos".E2_Off_Ev )
      R_Coil( "FIO_Esteira2" )
   END_RUNG
   // the same network as SCL:
   IF "Eventos".E2_On_Ev THEN "FIO_Esteira2" := TRUE; END_IF;
   IF "Eventos".E2_Off_Ev THEN "FIO_Esteira2" := FALSE; END_IF;
END_REGION

REGION Network 5: Esteira 3
   RUNG wire#powerrail
      Contact( "Eventos".E3_On_Ev )
      S_Coil( "FIO_Esteira3" )
   END_RUNG
   RUNG wire#powerrail
      Contact( "Eventos".E3_Off_Ev )
      R_Coil( "FIO_Esteira3" )
   END_RUNG
   // the same network as SCL:
   IF "Eventos".E3_On_Ev THEN "FIO_Esteira3" := TRUE; END_IF;
   IF "Eventos".E3_Off_Ev THEN "FIO_Esteira3" := FALSE; END_IF;
END_REGION

REGION Network 6: Esteira 4
   RUNG wire#powerrail
      Contact( "Eventos".E4_On_Ev )
      S_Coil( "FIO_Esteira4" )
   END_RUNG
   RUNG wire#powerrail
      Contact( "Eventos".E4_Off_Ev )
      R_Coil( "FIO_Esteira4" )
   END_RUNG
   // the same network as SCL:
   IF "Eventos".E4_On_Ev THEN "FIO_Esteira4" := TRUE; END_IF;
   IF "Eventos".E4_Off_Ev THEN "FIO_Esteira4" := FALSE; END_IF;
END_REGION
END_FUNCTION

ORGANIZATION_BLOCK "Main"   // OB1, LAD, ProgramCycle
TITLE = "Main Program Sweep (Cycle)"
{ S7_Optimized_Access := 'TRUE' }
VERSION : 0.1
   VAR_INPUT
      Initial_Call : Bool;   // Initial call of this OB
      Remanence : Bool;   // =True, if remanent data are available
   END_VAR
BEGIN

REGION Network 1
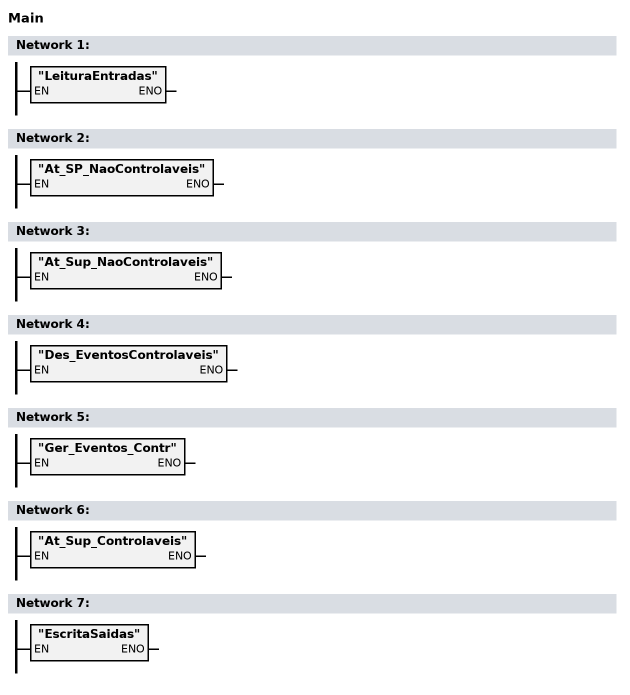
   RUNG wire#powerrail
      "LeituraEntradas"()
   END_RUNG
   // the same network as SCL:
   "LeituraEntradas"();
END_REGION

REGION Network 2
   RUNG wire#powerrail
      "At_SP_NaoControlaveis"()
   END_RUNG
   // the same network as SCL:
   "At_SP_NaoControlaveis"();
END_REGION

REGION Network 3
   RUNG wire#powerrail
      "At_Sup_NaoControlaveis"()
   END_RUNG
   // the same network as SCL:
   "At_Sup_NaoControlaveis"();
END_REGION

REGION Network 4
   RUNG wire#powerrail
      "Des_EventosControlaveis"()
   END_RUNG
   // the same network as SCL:
   "Des_EventosControlaveis"();
END_REGION

REGION Network 5
   RUNG wire#powerrail
      "Ger_Eventos_Contr"()
   END_RUNG
   // the same network as SCL:
   "Ger_Eventos_Contr"();
END_REGION

REGION Network 6
   RUNG wire#powerrail
      "At_Sup_Controlaveis"()
   END_RUNG
   // the same network as SCL:
   "At_Sup_Controlaveis"();
END_REGION

REGION Network 7
   RUNG wire#powerrail
      "EscritaSaidas"()
   END_RUNG
   // the same network as SCL:
   "EscritaSaidas"();
END_REGION
END_ORGANIZATION_BLOCK